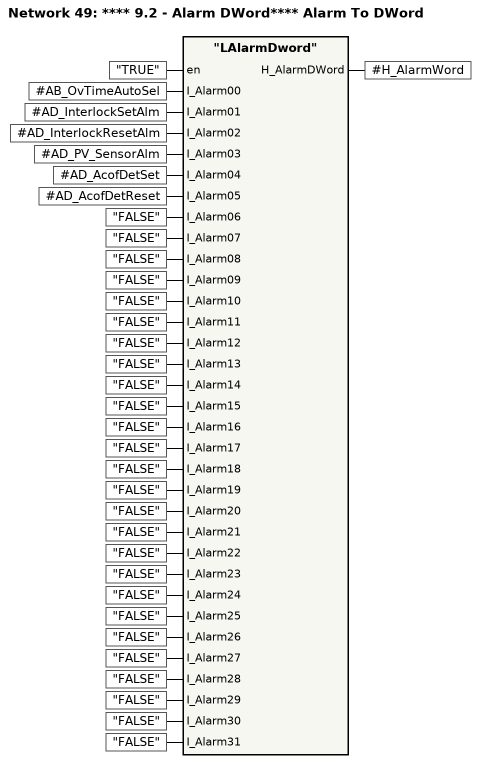
   IF "TRUE" THEN
       "LAlarmDword"(I_Alarm00 := #AB_OvTimeAutoSel,
                     I_Alarm01 := #AD_InterlockSetAlm,
                     I_Alarm02 := #AD_InterlockResetAlm,
                     I_Alarm03 := #AD_PV_SensorAlm,
                     I_Alarm04 := #AD_AcofDetSet,
                     I_Alarm05 := #AD_AcofDetReset,
                     I_Alarm06 := "FALSE",
                     I_Alarm07 := "FALSE",
                     I_Alarm08 := "FALSE",
                     I_Alarm09 := "FALSE",
                     I_Alarm10 := "FALSE",
                     I_Alarm11 := "FALSE",
                     I_Alarm12 := "FALSE",
                     I_Alarm13 := "FALSE",
                     I_Alarm14 := "FALSE",
                     I_Alarm15 := "FALSE",
                     I_Alarm16 := "FALSE",
                     I_Alarm17 := "FALSE",
                     I_Alarm18 := "FALSE",
                     I_Alarm19 := "FALSE",
                     I_Alarm20 := "FALSE",
                     I_Alarm21 := "FALSE",
                     I_Alarm22 := "FALSE",
                     I_Alarm23 := "FALSE",
                     I_Alarm24 := "FALSE",
                     I_Alarm25 := "FALSE",
                     I_Alarm26 := "FALSE",
                     I_Alarm27 := "FALSE",
                     I_Alarm28 := "FALSE",
                     I_Alarm29 := "FALSE",
                     I_Alarm30 := "FALSE",
                     I_Alarm31 := "FALSE",
                     H_AlarmDWord => #H_AlarmWord);
   END_IF;
END_REGION
END_FUNCTION_BLOCK

FUNCTION_BLOCK "LProcTimStrtStop"   // FB1735, FBD
TITLE = LProcTimeStartStop
{ S7_Optimized_Access := 'FALSE' }
AUTHOR : VCC
FAMILY : ProcEq
NAME : TimeStSt
VERSION : 1.0
// ================================================================================
// Module used to give a signal between 2 times with the calendar variable of PLC: 
// start - stop is defined by HMI
// ================================================================================
// stored: AutoNumber false, IsIECCheckEnabled false, SetENOAutomatically False, UDAEnableTagReadback false
   VAR_OUTPUT
      O_TimeActive { ExternalAccessible := 'False'; ExternalVisible := 'False'; ExternalWritable := 'False'} : Bool;   // Time active
      O_InverseTimeActive { ExternalAccessible := 'False'; ExternalVisible := 'False'; ExternalWritable := 'False'} : Bool;   // Inverse Time active
      H_IAnim { ExternalAccessible := 'False'; ExternalVisible := 'False'; ExternalWritable := 'False'} : Word;   // HMI Animation of the icon
   END_VAR
   VAR DB_SPECIFIC
      H_In : Struct   // HMI
         Start : Real := 9.0;   // Start time
         Stop : Real := 9.15;   // Stop time
      END_STRUCT;
      H_Out : Struct   // HMI
         Anim : Word;   // HMI Animation of the object
         DBnr : Int;   // HMI Animation DB number
      END_STRUCT;
      TimeActive { ExternalAccessible := 'False'; ExternalVisible := 'False'; ExternalWritable := 'False'} : Bool;   // Time active
      Start_Int { ExternalAccessible := 'False'; ExternalVisible := 'False'; ExternalWritable := 'False'} : Int := 900;   // Start integer
      Stop_Int { ExternalAccessible := 'False'; ExternalVisible := 'False'; ExternalWritable := 'False'} : Int := 915;   // Stort integer
      DBnr { ExternalAccessible := 'False'; ExternalVisible := 'False'; ExternalWritable := 'False'} : Int;   // HMI DB number
   END_VAR
BEGIN

NETWORK
TITLE = **** 1 - Inputs **** DB number
// DB number
      L     DINO;
      T     #DBnr;

NETWORK
TITLE = **** 4.4 - Machine status - Calculated **** Copy time from HMI to integer
// Copy time from HMI to integer
      L     #H_In.Start;  // Load Start time
      L     100.0;  // * 100
      *R;  // *
      RND;  // Conversion real to integer
      T     #Start_Int;  // Load start time of morning shift = Day 1

      L     #H_In.Stop;  // Load Start time of evening shift - Day 1
      L     100.0;  // * 100
      *R;  // *
      RND;  // Conversion real to integer
      T     #Stop_Int;  // Load start time of evening shift = Day 1


REGION Network 3: **** 4.4 - Machine status - Calculated **** Morning Shift of Day 1
   // Morning Shift of Day 1
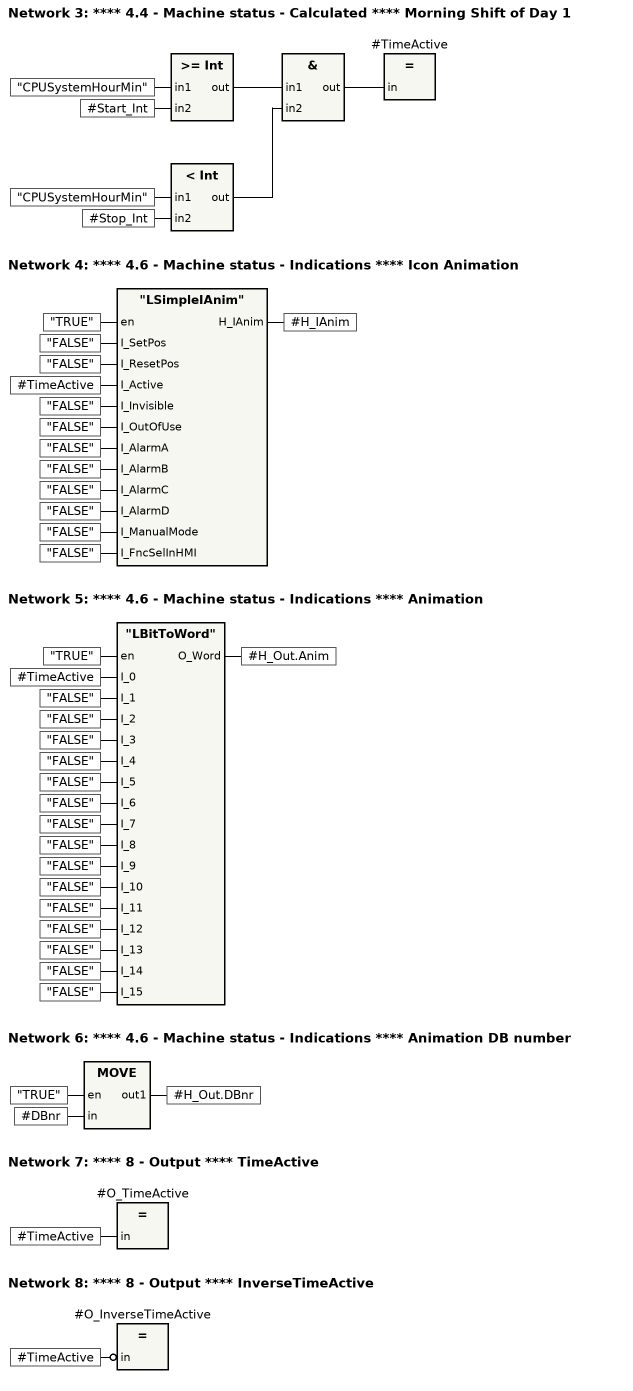
   #TimeActive := ("CPUSystemHourMin" >= #Start_Int) AND ("CPUSystemHourMin" < #Stop_Int);
END_REGION

REGION Network 4: **** 4.6 - Machine status - Indications **** Icon Animation
   // Icon Animation for HMI
   IF "TRUE" THEN
       "LSimpleIAnim"(I_SetPos := "FALSE",
                      I_ResetPos := "FALSE",
                      I_Active := #TimeActive,
                      I_Invisible := "FALSE",
                      I_OutOfUse := "FALSE",
                      I_AlarmA := "FALSE",
                      I_AlarmB := "FALSE",
                      I_AlarmC := "FALSE",
                      I_AlarmD := "FALSE",
                      I_ManualMode := "FALSE",
                      I_FncSelInHMI := "FALSE",
                      H_IAnim => #H_IAnim);
   END_IF;
END_REGION

REGION Network 5: **** 4.6 - Machine status - Indications **** Animation
   // Animation for HMI
   IF "TRUE" THEN
       "LBitToWord"(I_0 := #TimeActive,
                    I_1 := "FALSE",
                    I_2 := "FALSE",
                    I_3 := "FALSE",
                    I_4 := "FALSE",
                    I_5 := "FALSE",
                    I_6 := "FALSE",
                    I_7 := "FALSE",
                    I_8 := "FALSE",
                    I_9 := "FALSE",
                    I_10 := "FALSE",
                    I_11 := "FALSE",
                    I_12 := "FALSE",
                    I_13 := "FALSE",
                    I_14 := "FALSE",
                    I_15 := "FALSE",
                    O_Word => #H_Out.Anim);
   END_IF;
END_REGION

REGION Network 6: **** 4.6 - Machine status - Indications **** Animation DB number
   // Animation DB number
   IF "TRUE" THEN #H_Out.DBnr := #DBnr; END_IF;
END_REGION

REGION Network 7: **** 8 - Output **** TimeActive
   // TimeActive
   #O_TimeActive := #TimeActive;
END_REGION

REGION Network 8: **** 8 - Output **** InverseTimeActive
   // InverseTimeActive
   #O_InverseTimeActive := NOT #TimeActive;
END_REGION
END_FUNCTION_BLOCK

FUNCTION_BLOCK "LProcGeneralFunc"   // FB1738, FBD
TITLE = LProcGeneralFunc
{ S7_Optimized_Access := 'TRUE' }
AUTHOR : VCC
FAMILY : Control
NAME : Genfunc
VERSION : 0.1
// ================================================================================
// This module handles General Reverse Switch, General High Speed and Lamptest.
// It will also give the user and 8 bit interface for project specific functions.
// ================================================================================
// stored: AutoNumber false, IsIECCheckEnabled false, IsRetainMemResEnabled false, MemoryReserve 100, SetENOAutomatically False, UDAEnableTagReadback false
   VAR_INPUT
      I_GenRevSw { ExternalAccessible := 'False'; ExternalVisible := 'False'; ExternalWritable := 'False'} : Bool;   // General reverse switch
      I_GenHighSpeed { ExternalAccessible := 'False'; ExternalVisible := 'False'; ExternalWritable := 'False'} : Bool;   // General high speed
      I_Lamptest { ExternalAccessible := 'False'; ExternalVisible := 'False'; ExternalWritable := 'False'} : Bool;   // Lamptest PB
      I_ManualMode { ExternalAccessible := 'False'; ExternalVisible := 'False'; ExternalWritable := 'False'} : Bool := TRUE;   // Manual mode active
      I_LamptestSec { ExternalAccessible := 'False'; ExternalVisible := 'False'; ExternalWritable := 'False'} : Int := 60;   // The number of seconds that Lamptest will be on (Sec)
   END_VAR
   VAR_OUTPUT
      O_GeneralFunc : Word;   // General functions
      O_Lamptest { ExternalAccessible := 'False'; ExternalVisible := 'False'; ExternalWritable := 'False'} : Bool;   // Lamptest
      O_LamptestSteady { ExternalAccessible := 'False'; ExternalVisible := 'False'; ExternalWritable := 'False'} : Bool;   // Lamptest always on
      O_GenHighSpeed { ExternalAccessible := 'False'; ExternalVisible := 'False'; ExternalWritable := 'False'} : Bool;   // General High Speed
      O_GenRevSwitch { ExternalAccessible := 'False'; ExternalVisible := 'False'; ExternalWritable := 'False'} : Bool;   // Reverse Switch
      O_GenReverseAlarm { ExternalAccessible := 'False'; ExternalVisible := 'False'; ExternalWritable := 'False'} : Bool;   // Alarm when general reverse switch is ON while NOT in Manual mode
   END_VAR
   VAR DB_SPECIFIC
      H_HMIGenFuncCmd : Word;   // General function commands from HMI
      AutoMode { ExternalAccessible := 'False'; ExternalVisible := 'False'; ExternalWritable := 'False'} : Bool;   // Auto mode
      AutoSel { ExternalAccessible := 'False'; ExternalVisible := 'False'; ExternalWritable := 'False'} : Bool;   // Auto is selected
      AlarmAB { ExternalAccessible := 'False'; ExternalVisible := 'False'; ExternalWritable := 'False'} : Bool;   // Alarm A or B is active
      HMIGenHighSpeed { ExternalAccessible := 'False'; ExternalVisible := 'False'; ExternalWritable := 'False'} : Bool;   // General High Speed for manual movement
      HMILamptest { ExternalAccessible := 'False'; ExternalVisible := 'False'; ExternalWritable := 'False'} : Bool;   // Lamptest
      GenHighSpeedSelected { ExternalAccessible := 'False'; ExternalVisible := 'False'; ExternalWritable := 'False'} : Bool;   // General high speed is selected
      LamptestSelected : Bool;   // Lamptest is selected
      PulseLamptest { ExternalAccessible := 'False'; ExternalVisible := 'False'; ExternalWritable := 'False'} : Bool;   // Pulse for lamptest
      PulseGenHighSpeed { ExternalAccessible := 'False'; ExternalVisible := 'False'; ExternalWritable := 'False'} : Bool;   // Pulse General high speed
      TimerLamptest { ExternalAccessible := 'False'; ExternalVisible := 'False'; ExternalWritable := 'False'} : Bool;   // Timer for Lamptest
      LamptestSec { ExternalAccessible := 'False'; ExternalVisible := 'False'; ExternalWritable := 'False'} : DInt;   // Lamptest on for xxx milliesec
      LamptestMillieSec { ExternalAccessible := 'False'; ExternalVisible := 'False'; ExternalWritable := 'False'} : DInt;   // Converted value
   END_VAR
   VAR
      TimerLampTestSel { ExternalAccessible := 'False'; ExternalVisible := 'False'; ExternalWritable := 'False'; S7_SetPoint := 'True'} : "LTimer";
   END_VAR
   VAR_TEMP
      SetLamptest : Bool;   // Set Lamptest
      ResetLamptest : Bool;   // Reset Lamptest
      ElapseTime : DInt;   // Elapse time for Lamptest
   END_VAR
   VAR_TEMP   // added for the SCL form of the ladder/FBD networks
      _w1 : Bool;
      _w2 : Bool;
   END_VAR
BEGIN

REGION Network 1: **** 1 - Inputs **** Extract the general functions from HMI
   // Extract the general functions from HMI
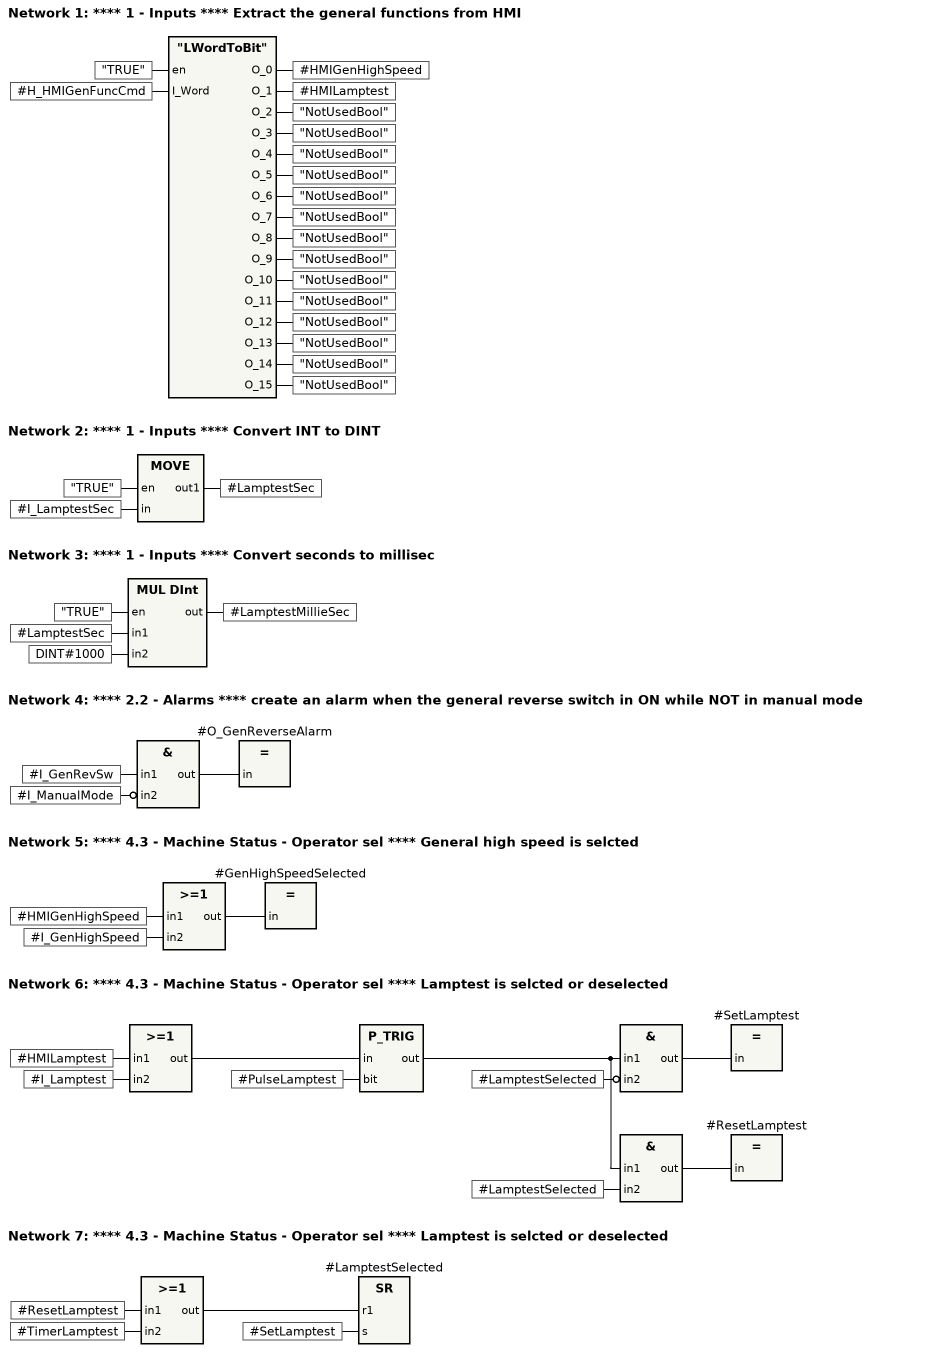
   IF "TRUE" THEN
       "LWordToBit"(I_Word := #H_HMIGenFuncCmd,
                    O_0 => #HMIGenHighSpeed,
                    O_1 => #HMILamptest,
                    O_2 => "NotUsedBool",
                    O_3 => "NotUsedBool",
                    O_4 => "NotUsedBool",
                    O_5 => "NotUsedBool",
                    O_6 => "NotUsedBool",
                    O_7 => "NotUsedBool",
                    O_8 => "NotUsedBool",
                    O_9 => "NotUsedBool",
                    O_10 => "NotUsedBool",
                    O_11 => "NotUsedBool",
                    O_12 => "NotUsedBool",
                    O_13 => "NotUsedBool",
                    O_14 => "NotUsedBool",
                    O_15 => "NotUsedBool");
   END_IF;
END_REGION

REGION Network 2: **** 1 - Inputs **** Convert INT to DINT
   // Convert INT to DINT
   IF "TRUE" THEN #LamptestSec := #I_LamptestSec; END_IF;
END_REGION

REGION Network 3: **** 1 - Inputs **** Convert seconds to millisec
   // Convert seconds to millisec
   IF "TRUE" THEN #LamptestMillieSec := #LamptestSec * DINT#1000; END_IF;
END_REGION

REGION Network 4: **** 2.2 - Alarms **** create an alarm when the general reverse switch in ON while NOT in manual mode
   // create an alarm when the general reverse switch in ON while NOT in manual mode
   #O_GenReverseAlarm := #I_GenRevSw AND NOT #I_ManualMode;
END_REGION

REGION Network 5: **** 4.3 - Machine Status - Operator sel **** General high speed is selcted
   // General high speed is selcted
   #GenHighSpeedSelected := #HMIGenHighSpeed OR #I_GenHighSpeed;
END_REGION

REGION Network 6: **** 4.3 - Machine Status - Operator sel **** Lamptest is selcted or deselected
   // Lamptest is selcted or deselected
   #_w1 := #HMILamptest OR #I_Lamptest;
   #_w2 := #_w1 AND NOT #PulseLamptest;   // rising edge
   #PulseLamptest := #_w1;
   #SetLamptest := #_w2 AND NOT #LamptestSelected;
   #ResetLamptest := #_w2 AND #LamptestSelected;
END_REGION

REGION Network 7: **** 4.3 - Machine Status - Operator sel **** Lamptest is selcted or deselected
   // Lamptest is selcted or deselected
   IF #SetLamptest THEN
       #LamptestSelected := TRUE;   // SR flip-flop
   END_IF;
   IF #ResetLamptest OR #TimerLamptest THEN #LamptestSelected := FALSE; END_IF;
END_REGION

REGION Network 8: **** 4.3 - Machine Status - Operator sel **** Timer for Lamptest
   // Timer for Lamptest
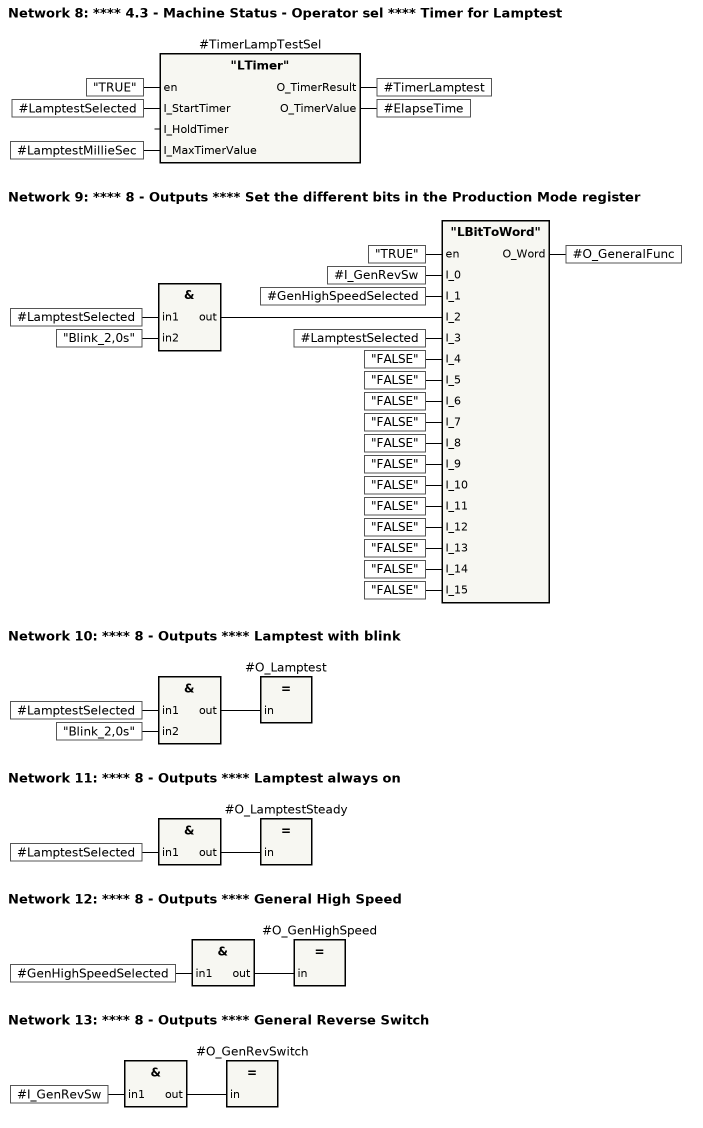
   IF "TRUE" THEN
       #TimerLampTestSel(I_StartTimer := #LamptestSelected,   // "LTimer"
                         I_MaxTimerValue := #LamptestMillieSec,
                         O_TimerResult => #TimerLamptest,
                         O_TimerValue => #ElapseTime);
   END_IF;
END_REGION

REGION Network 9: **** 8 - Outputs **** Set the different bits in the Production Mode register
   // Set the different bits in the Production Mode register
   IF "TRUE" THEN
       "LBitToWord"(I_0 := #I_GenRevSw,
                    I_1 := #GenHighSpeedSelected,
                    I_2 := #LamptestSelected AND "Blink_2,0s",
                    I_3 := #LamptestSelected,
                    I_4 := "FALSE",
                    I_5 := "FALSE",
                    I_6 := "FALSE",
                    I_7 := "FALSE",
                    I_8 := "FALSE",
                    I_9 := "FALSE",
                    I_10 := "FALSE",
                    I_11 := "FALSE",
                    I_12 := "FALSE",
                    I_13 := "FALSE",
                    I_14 := "FALSE",
                    I_15 := "FALSE",
                    O_Word => #O_GeneralFunc);
   END_IF;
END_REGION

REGION Network 10: **** 8 - Outputs **** Lamptest with blink
   // Lamptest with blink
   #O_Lamptest := #LamptestSelected AND "Blink_2,0s";
END_REGION

REGION Network 11: **** 8 - Outputs **** Lamptest always on
   // Lamptest always on
   #O_LamptestSteady := #LamptestSelected;
END_REGION

REGION Network 12: **** 8 - Outputs **** General High Speed
   // General High Speed
   #O_GenHighSpeed := #GenHighSpeedSelected;
END_REGION

REGION Network 13: **** 8 - Outputs **** General Reverse Switch
   // General Reverse Switch
   #O_GenRevSwitch := #I_GenRevSw;
END_REGION
END_FUNCTION_BLOCK

FUNCTION_BLOCK "LProcPAC"   // FB1740, FBD
TITLE = LProcPAC
{ S7_Optimized_Access := 'TRUE' }
AUTHOR : CSTAAL
VERSION : 0.1
// This module handles the power measuring device
// stored: AutoNumber false, IsIECCheckEnabled false, IsRetainMemResEnabled false, MemoryReserve 100, SetENOAutomatically False, UDAEnableTagReadback false
   VAR_INPUT
      I_HWSubModule { ExternalAccessible := 'False'; ExternalVisible := 'False'; ExternalWritable := 'False'} : HW_SUBMODULE;   // Connection with Hardware Sub Module
   END_VAR
   VAR_OUTPUT
      O_ControlBytes { ExternalAccessible := 'False'; ExternalVisible := 'False'; ExternalWritable := 'False'} : Word;   // Control Bytes for the PAC
      O_AlarmA { ExternalAccessible := 'False'; ExternalVisible := 'False'; ExternalWritable := 'False'} : Bool;   // Alarm A
      O_AlarmB { ExternalAccessible := 'False'; ExternalVisible := 'False'; ExternalWritable := 'False'} : Bool;   // Alarm B
      O_AlarmC { ExternalAccessible := 'False'; ExternalVisible := 'False'; ExternalWritable := 'False'} : Bool;   // Alarm C
      O_AlarmD { ExternalAccessible := 'False'; ExternalVisible := 'False'; ExternalWritable := 'False'} : Bool;   // Alarm D
      O_AlarmABCondition { ExternalAccessible := 'False'; ExternalVisible := 'False'; ExternalWritable := 'False'} : Bool;   // Alarms resetable
      H_IAnim { ExternalAccessible := 'False'; ExternalVisible := 'False'; ExternalWritable := 'False'} : Word;   // Animation bits to Icon in WinCC
      H_AlarmWord { ExternalAccessible := 'False'; ExternalVisible := 'False'; ExternalWritable := 'False'} : DWord;   // Alarm Word
   END_VAR
   VAR DB_SPECIFIC
      Cmd { ExternalAccessible := 'False'; ExternalVisible := 'False'; ExternalWritable := 'False'} : Struct   // Command (copied from HMI Command) / Command
         Reset_min_max_Data { ExternalAccessible := 'False'; ExternalVisible := 'False'; ExternalWritable := 'False'} : Bool := FALSE;   // 0 / Reset_min_max_Data
         Reset_Energy_Meter { ExternalAccessible := 'False'; ExternalVisible := 'False'; ExternalWritable := 'False'} : Bool := FALSE;   // 1 / Reset_Energy_Meter
      END_STRUCT;
   END_VAR
   VAR
      C_UnitAmps { ExternalAccessible := 'False'; ExternalVisible := 'False'; ExternalWritable := 'False'} : Int;   // Unit Amps (1 = mA; 2 = kA)
      C_UnitVolts { ExternalAccessible := 'False'; ExternalVisible := 'False'; ExternalWritable := 'False'} : Int;   // Unit Volts (1 = mV; 2 = V)
      C_UnitWatts { ExternalAccessible := 'False'; ExternalVisible := 'False'; ExternalWritable := 'False'} : Int;   // Unit Watts (1 = W; 2 = kW)
      Units { ExternalAccessible := 'False'; ExternalVisible := 'False'; ExternalWritable := 'False'} : Struct   // Units
         "Amps-mA" { ExternalAccessible := 'False'; ExternalVisible := 'False'; ExternalWritable := 'False'} : Bool;   // Amps in mA
         "Amps-kA" { ExternalAccessible := 'False'; ExternalVisible := 'False'; ExternalWritable := 'False'} : Bool;   // Amps in kA
         "Volts-mV" { ExternalAccessible := 'False'; ExternalVisible := 'False'; ExternalWritable := 'False'} : Bool;   // Volts in mV
         "Volts-kV" { ExternalAccessible := 'False'; ExternalVisible := 'False'; ExternalWritable := 'False'} : Bool;   // Volts in kV
         "Watts-W" { ExternalAccessible := 'False'; ExternalVisible := 'False'; ExternalWritable := 'False'} : Bool;   // Watts in W
         "Watts-kW" { ExternalAccessible := 'False'; ExternalVisible := 'False'; ExternalWritable := 'False'} : Bool;   // Watts in kW
      END_STRUCT;
      H_HMICmd : Word;   // HMI Command
   END_VAR
   VAR DB_SPECIFIC
      H_Out : Struct   // HMI
         Anim : Word;   // HMI Animation of the object
         DBnr : Int;   // HMI Animation DB number
         U12 : Real;   // Voltage L1-L2
         U23 : Real;   // Voltage L2-L3
         U31 : Real;   // Voltage L3-L1
         U12Max : Real;   // MAX Voltage L1-L2
         U23Max : Real;   // MAX Voltage L2-L3
         U31Max : Real;   // MAX Voltage L3-L1
         UL1 : Real;   // UL1
         UL2 : Real;   // UL2
         UL3 : Real;   // UL3
         UL1Max : Real;   // MAX Voltage L1
         UL2Max : Real;   // MAX Voltage L2
         UL3Max : Real;   // MAX Voltage L3
         I1 : Real;   // Current L1
         I2 : Real;   // Current L2
         I3 : Real;   // Current L3
         I1Max : Real;   // MAX Current L1
         I2Max : Real;   // MAX Current L2
         I3Max : Real;   // MAX Current L3
         PTotal : Real;   // Total active power
         PTotalMax : Real;   // Total MAX active power
      END_STRUCT;
   END_VAR
   VAR
      AlarmA { ExternalAccessible := 'False'; ExternalVisible := 'False'; ExternalWritable := 'False'} : Bool;   // Alarm A
      AlarmB { ExternalAccessible := 'False'; ExternalVisible := 'False'; ExternalWritable := 'False'} : Bool;   // Alarm B
      AlarmC { ExternalAccessible := 'False'; ExternalVisible := 'False'; ExternalWritable := 'False'} : Bool;   // Alarm C
      AlarmD { ExternalAccessible := 'False'; ExternalVisible := 'False'; ExternalWritable := 'False'} : Bool;   // Alarm D
      AlarmABCondition { ExternalAccessible := 'False'; ExternalVisible := 'False'; ExternalWritable := 'False'} : Bool;   // Alarm AB condition
   END_VAR
   VAR DB_SPECIFIC
      DBnr { ExternalAccessible := 'False'; ExternalVisible := 'False'; ExternalWritable := 'False'} : Int;   // HMI DB number
   END_VAR
   VAR
      _PACDriver { ExternalAccessible := 'False'; ExternalVisible := 'False'; ExternalWritable := 'False'} : "LProcPAC-Driver";   // FB
      _PACVisu { ExternalAccessible := 'False'; ExternalVisible := 'False'; ExternalWritable := 'False'} : "LProcPAC-Visu";   // FB
   END_VAR
   VAR_TEMP
      ControlBytes : Word;   // Control Bytes for the PAC
      L12 : Real;   // Temporary test variable
      L23 : Real;   // Temporary test variable
      L31 : Real;   // Temporary test variable
   END_VAR
   VAR_TEMP   // added for the SCL form of the ladder/FBD networks
      _w1 : Bool;
   END_VAR
BEGIN

NETWORK
TITLE = **** 1 - Inputs **** DB number
// DB number
      L     DINO;
      T     #DBnr;

REGION Network 2: **** 1 - Inputs **** HMI Commands
   // HMI Commands
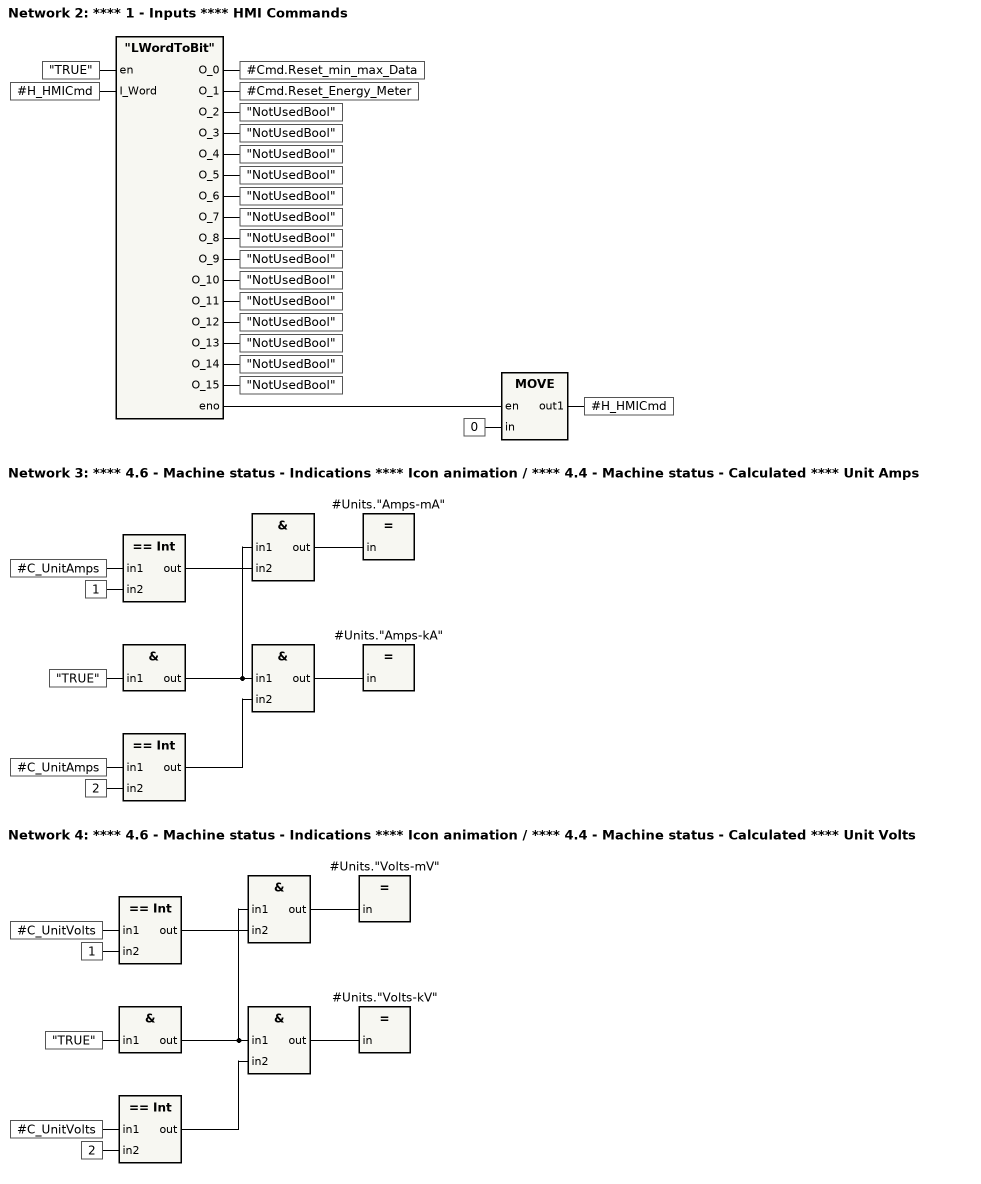
   "LWordToBit"(EN := "TRUE",
                I_Word := #H_HMICmd,
                O_0 => #Cmd.Reset_min_max_Data,
                O_1 => #Cmd.Reset_Energy_Meter,
                O_2 => "NotUsedBool",
                O_3 => "NotUsedBool",
                O_4 => "NotUsedBool",
                O_5 => "NotUsedBool",
                O_6 => "NotUsedBool",
                O_7 => "NotUsedBool",
                O_8 => "NotUsedBool",
                O_9 => "NotUsedBool",
                O_10 => "NotUsedBool",
                O_11 => "NotUsedBool",
                O_12 => "NotUsedBool",
                O_13 => "NotUsedBool",
                O_14 => "NotUsedBool",
                O_15 => "NotUsedBool",
                ENO => #_w1);
   IF #_w1 THEN #H_HMICmd := 0; END_IF;
END_REGION

REGION Network 3: **** 4.6 - Machine status - Indications **** Icon animation / **** 4.4 - Machine status - Calculated **** Unit Amps
   // Icon animation to WinCC / Unit Amps
   #Units."Amps-mA" := "TRUE" AND (#C_UnitAmps = 1);
   #Units."Amps-kA" := "TRUE" AND (#C_UnitAmps = 2);
END_REGION

REGION Network 4: **** 4.6 - Machine status - Indications **** Icon animation / **** 4.4 - Machine status - Calculated **** Unit Volts
   // Icon animation to WinCC / Unit Volts
   #Units."Volts-mV" := "TRUE" AND (#C_UnitVolts = 1);
   #Units."Volts-kV" := "TRUE" AND (#C_UnitVolts = 2);
END_REGION

REGION Network 5: **** 4.6 - Machine status - Indications **** Icon animation / **** 4.4 - Machine status - Calculated **** Unit Watts
   // Icon animation to WinCC / Unit Watts
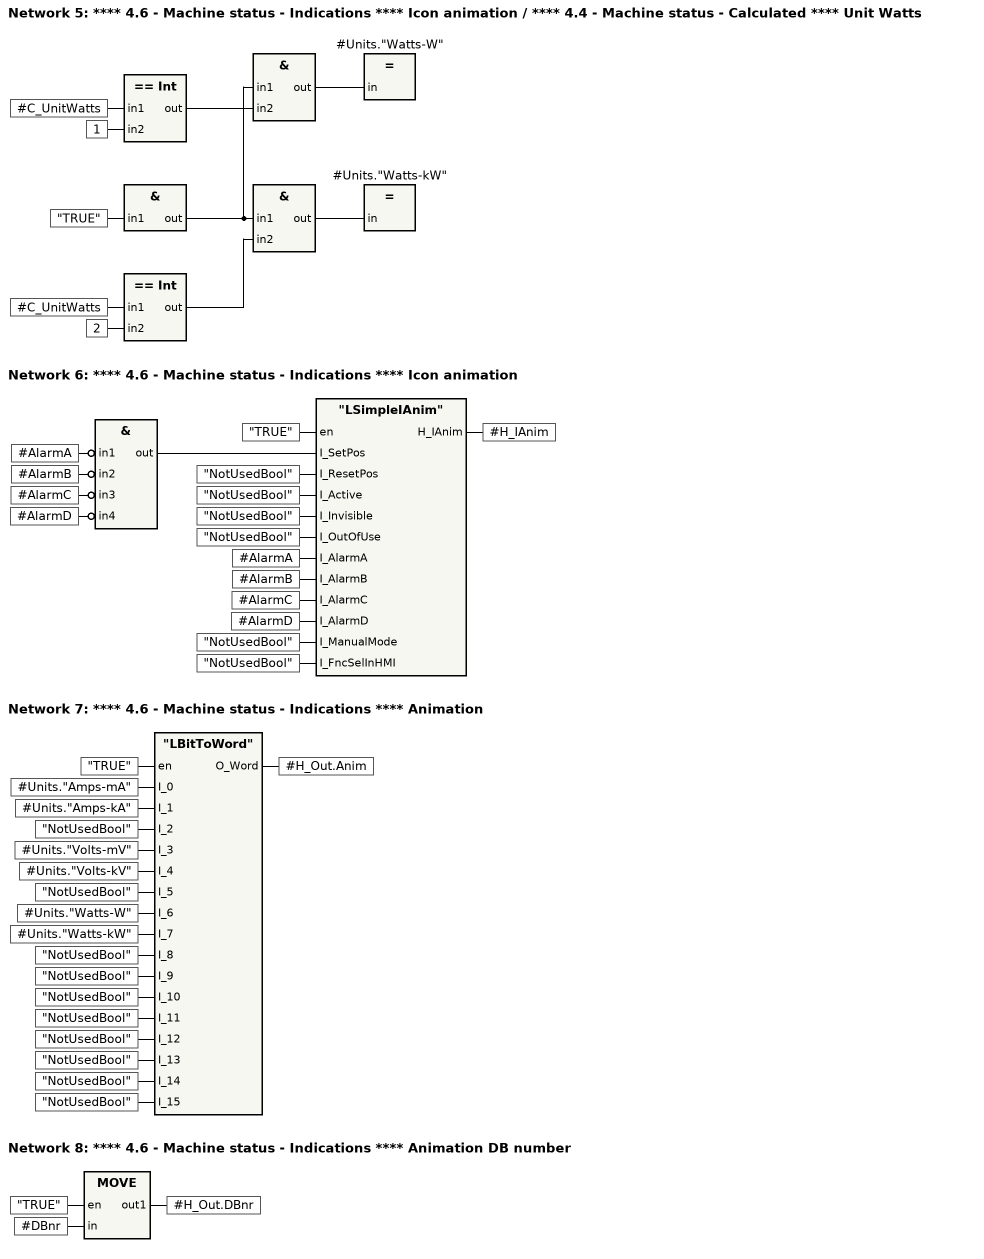
   #Units."Watts-W" := "TRUE" AND (#C_UnitWatts = 1);
   #Units."Watts-kW" := "TRUE" AND (#C_UnitWatts = 2);
END_REGION

REGION Network 6: **** 4.6 - Machine status - Indications **** Icon animation
   // Icon animation to WinCC / Icon animation
   IF "TRUE" THEN
       "LSimpleIAnim"(I_SetPos := NOT #AlarmA AND NOT #AlarmB AND NOT #AlarmC AND NOT #AlarmD,
                      I_ResetPos := "NotUsedBool",
                      I_Active := "NotUsedBool",
                      I_Invisible := "NotUsedBool",
                      I_OutOfUse := "NotUsedBool",
                      I_AlarmA := #AlarmA,
                      I_AlarmB := #AlarmB,
                      I_AlarmC := #AlarmC,
                      I_AlarmD := #AlarmD,
                      I_ManualMode := "NotUsedBool",
                      I_FncSelInHMI := "NotUsedBool",
                      H_IAnim => #H_IAnim);
   END_IF;
END_REGION

REGION Network 7: **** 4.6 - Machine status - Indications **** Animation
   // Animation
   IF "TRUE" THEN
       "LBitToWord"(I_0 := #Units."Amps-mA",
                    I_1 := #Units."Amps-kA",
                    I_2 := "NotUsedBool",
                    I_3 := #Units."Volts-mV",
                    I_4 := #Units."Volts-kV",
                    I_5 := "NotUsedBool",
                    I_6 := #Units."Watts-W",
                    I_7 := #Units."Watts-kW",
                    I_8 := "NotUsedBool",
                    I_9 := "NotUsedBool",
                    I_10 := "NotUsedBool",
                    I_11 := "NotUsedBool",
                    I_12 := "NotUsedBool",
                    I_13 := "NotUsedBool",
                    I_14 := "NotUsedBool",
                    I_15 := "NotUsedBool",
                    O_Word => #H_Out.Anim);
   END_IF;
END_REGION

REGION Network 8: **** 4.6 - Machine status - Indications **** Animation DB number
   // Animation DB number
   IF "TRUE" THEN #H_Out.DBnr := #DBnr; END_IF;
END_REGION

REGION Network 9: **** 7.1 SubModules - Non Machine **** Method 2: PAC3200 Driver
   // PAC3200 Driver
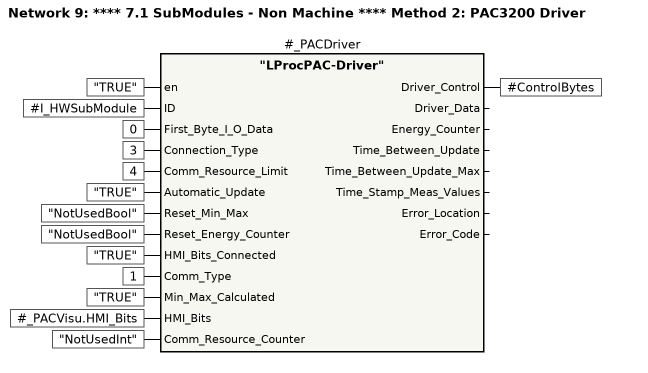
   IF "TRUE" THEN
       #_PACDriver(ID := #I_HWSubModule,   // "LProcPAC-Driver"
                   First_Byte_I_O_Data := 0,
                   Connection_Type := 3,
                   Comm_Resource_Limit := 4,
                   Automatic_Update := "TRUE",
                   Reset_Min_Max := "NotUsedBool",
                   Reset_Energy_Counter := "NotUsedBool",
                   HMI_Bits_Connected := "TRUE",
                   Comm_Type := 1,
                   Min_Max_Calculated := "TRUE",
                   HMI_Bits := #_PACVisu.HMI_Bits,
                   Comm_Resource_Counter := "NotUsedInt",
                   Driver_Control => #ControlBytes);
   END_IF;
END_REGION

REGION Network 10: **** 7.1 SubModules - Non Machine **** Method 2: PAC3200 Visualisation
   // PAC3200 Visualisation
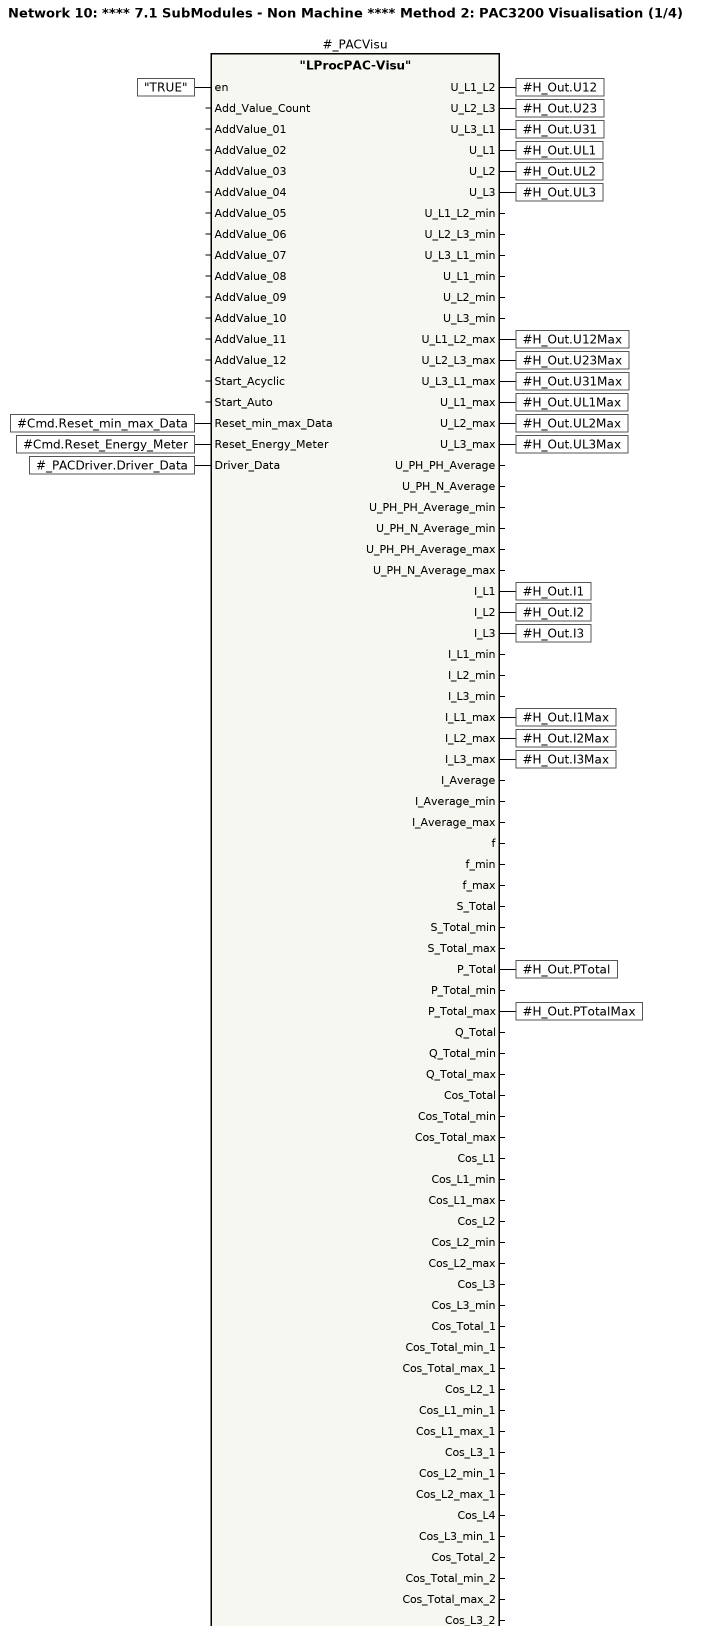
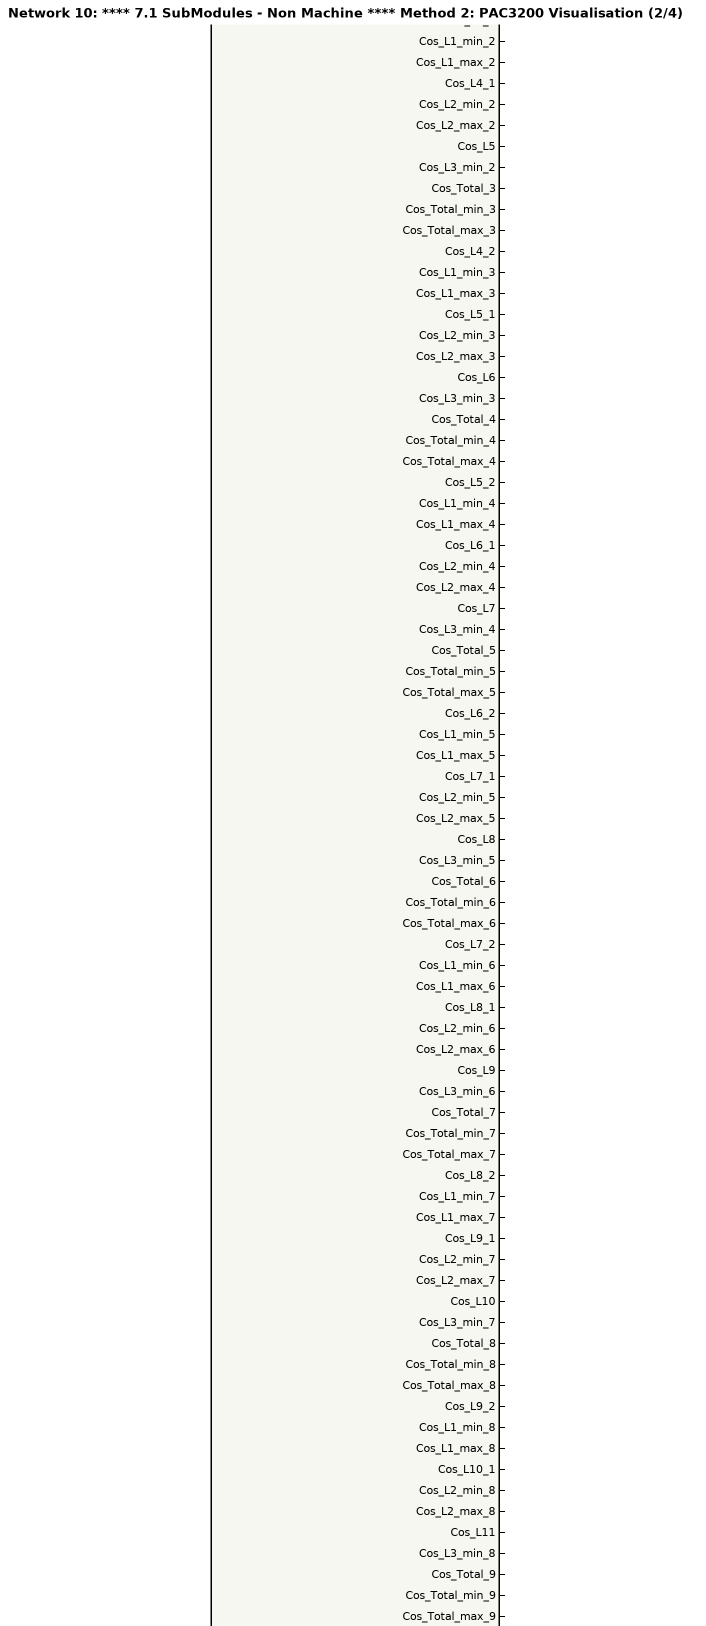
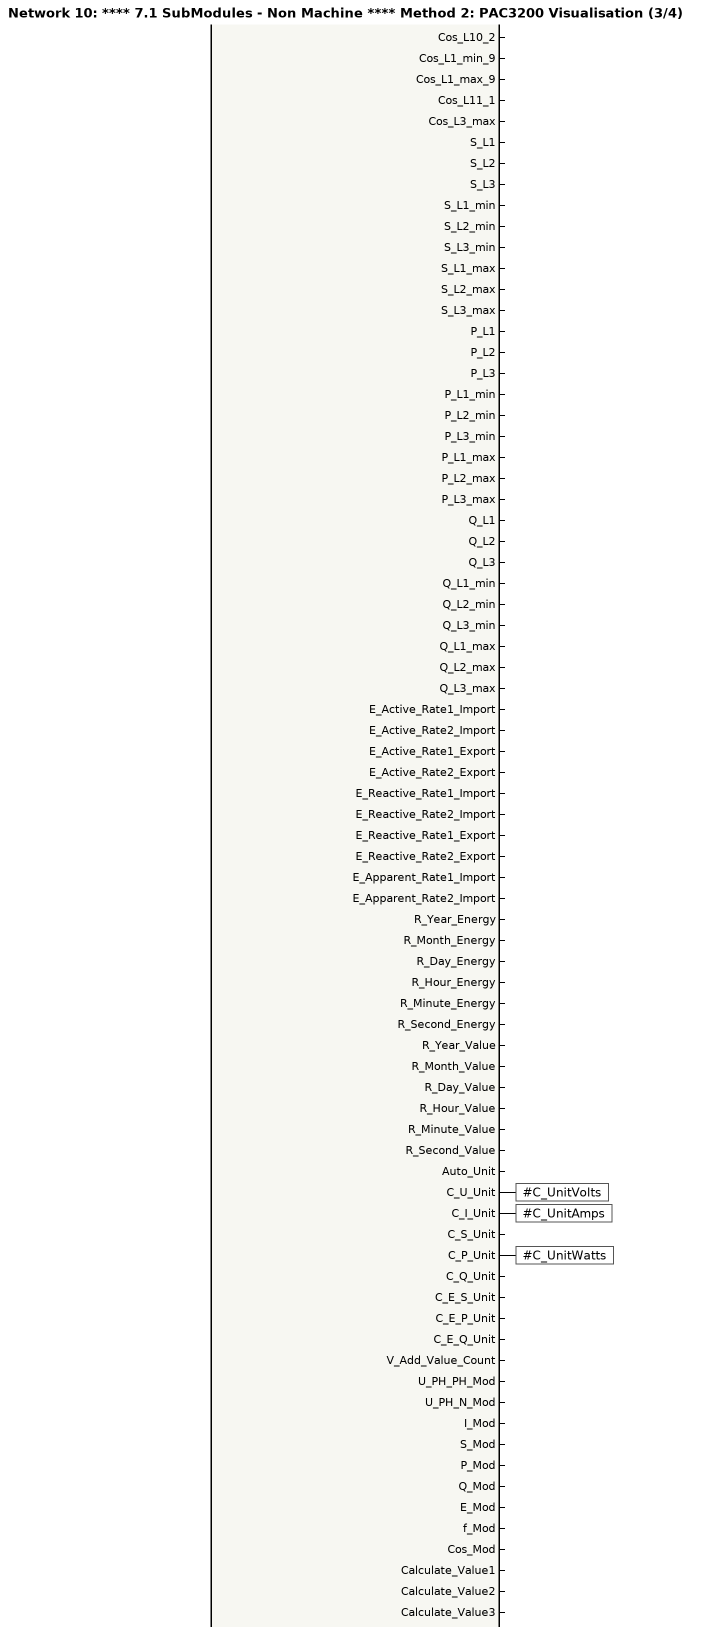
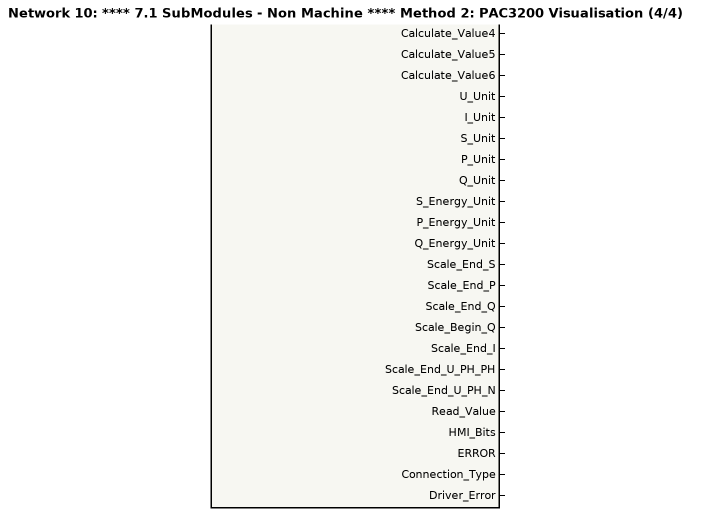
   IF "TRUE" THEN
       #_PACVisu(Reset_min_max_Data := #Cmd.Reset_min_max_Data,   // "LProcPAC-Visu"
                 Reset_Energy_Meter := #Cmd.Reset_Energy_Meter,
                 Driver_Data := #_PACDriver.Driver_Data,
                 U_L1_L2 => #H_Out.U12,
                 U_L2_L3 => #H_Out.U23,
                 U_L3_L1 => #H_Out.U31,
                 U_L1 => #H_Out.UL1,
                 U_L2 => #H_Out.UL2,
                 U_L3 => #H_Out.UL3,
                 U_L1_L2_max => #H_Out.U12Max,
                 U_L2_L3_max => #H_Out.U23Max,
                 U_L3_L1_max => #H_Out.U31Max,
                 U_L1_max => #H_Out.UL1Max,
                 U_L2_max => #H_Out.UL2Max,
                 U_L3_max => #H_Out.UL3Max,
                 I_L1 => #H_Out.I1,
                 I_L2 => #H_Out.I2,
                 I_L3 => #H_Out.I3,
                 I_L1_max => #H_Out.I1Max,
                 I_L2_max => #H_Out.I2Max,
                 I_L3_max => #H_Out.I3Max,
                 P_Total => #H_Out.PTotal,
                 P_Total_max => #H_Out.PTotalMax,
                 C_U_Unit => #C_UnitVolts,
                 C_I_Unit => #C_UnitAmps,
                 C_P_Unit => #C_UnitWatts);
   END_IF;
END_REGION

REGION Network 11: *** 8 - Outputs **** Control Bytes PAC
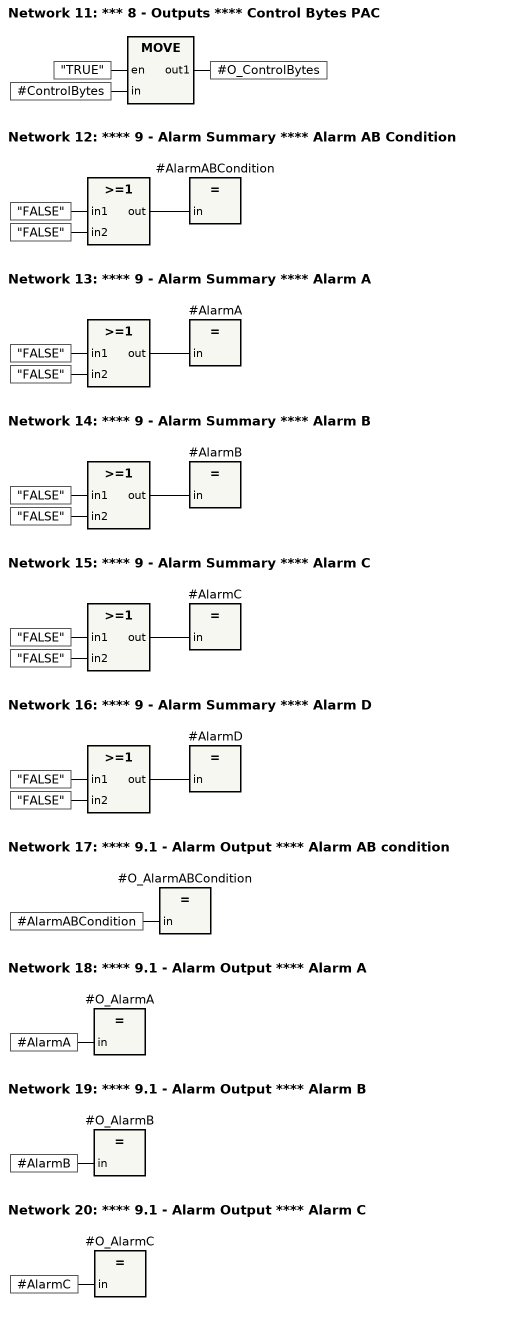
   IF "TRUE" THEN #O_ControlBytes := #ControlBytes; END_IF;
END_REGION

REGION Network 12: **** 9 - Alarm Summary **** Alarm AB Condition
   #AlarmABCondition := "FALSE" OR "FALSE";
END_REGION

REGION Network 13: **** 9 - Alarm Summary **** Alarm A
   #AlarmA := "FALSE" OR "FALSE";
END_REGION

REGION Network 14: **** 9 - Alarm Summary **** Alarm B
   #AlarmB := "FALSE" OR "FALSE";
END_REGION

REGION Network 15: **** 9 - Alarm Summary **** Alarm C
   #AlarmC := "FALSE" OR "FALSE";
END_REGION

REGION Network 16: **** 9 - Alarm Summary **** Alarm D
   #AlarmD := "FALSE" OR "FALSE";
END_REGION

REGION Network 17: **** 9.1 - Alarm Output **** Alarm AB condition
   // Alarm AB condition
   #O_AlarmABCondition := #AlarmABCondition;
END_REGION

REGION Network 18: **** 9.1 - Alarm Output **** Alarm A
   // Output Alarm A
   #O_AlarmA := #AlarmA;
END_REGION

REGION Network 19: **** 9.1 - Alarm Output **** Alarm B
   // Output Alarm B
   #O_AlarmB := #AlarmB;
END_REGION

REGION Network 20: **** 9.1 - Alarm Output **** Alarm C
   // Output Alarm A
   #O_AlarmC := #AlarmC;
END_REGION

REGION Network 21: **** 9.1 - Alarm Output **** Alarm D
   // Output Alarm D
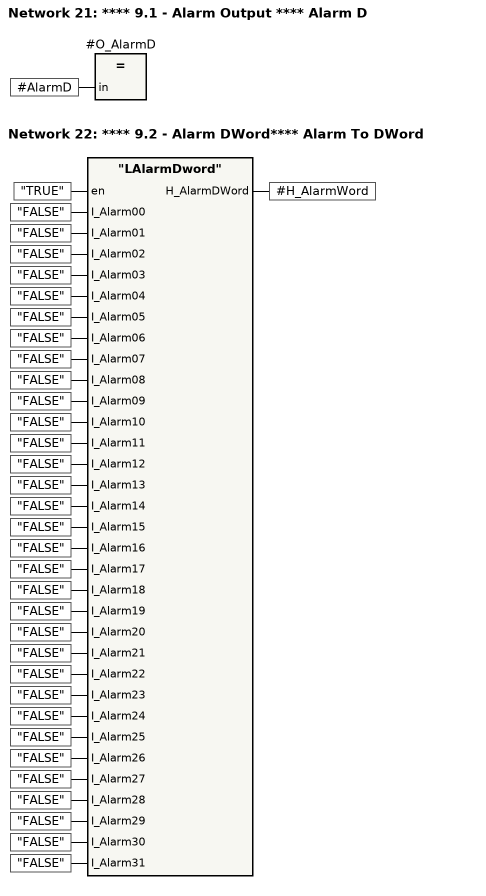
   #O_AlarmD := #AlarmD;
END_REGION

REGION Network 22: **** 9.2 - Alarm DWord**** Alarm To DWord
   // Alarm Word
   IF "TRUE" THEN
       "LAlarmDword"(I_Alarm00 := "FALSE",
                     I_Alarm01 := "FALSE",
                     I_Alarm02 := "FALSE",
                     I_Alarm03 := "FALSE",
                     I_Alarm04 := "FALSE",
                     I_Alarm05 := "FALSE",
                     I_Alarm06 := "FALSE",
                     I_Alarm07 := "FALSE",
                     I_Alarm08 := "FALSE",
                     I_Alarm09 := "FALSE",
                     I_Alarm10 := "FALSE",
                     I_Alarm11 := "FALSE",
                     I_Alarm12 := "FALSE",
                     I_Alarm13 := "FALSE",
                     I_Alarm14 := "FALSE",
                     I_Alarm15 := "FALSE",
                     I_Alarm16 := "FALSE",
                     I_Alarm17 := "FALSE",
                     I_Alarm18 := "FALSE",
                     I_Alarm19 := "FALSE",
                     I_Alarm20 := "FALSE",
                     I_Alarm21 := "FALSE",
                     I_Alarm22 := "FALSE",
                     I_Alarm23 := "FALSE",
                     I_Alarm24 := "FALSE",
                     I_Alarm25 := "FALSE",
                     I_Alarm26 := "FALSE",
                     I_Alarm27 := "FALSE",
                     I_Alarm28 := "FALSE",
                     I_Alarm29 := "FALSE",
                     I_Alarm30 := "FALSE",
                     I_Alarm31 := "FALSE",
                     H_AlarmDWord => #H_AlarmWord);
   END_IF;
END_REGION
END_FUNCTION_BLOCK

FUNCTION_BLOCK "LProcPAC-Driver"   // FB1741, SCL
TITLE = LProcPAC-Driver
{ S7_Optimized_Access := 'FALSE' }
AUTHOR : CSTAAL
VERSION : 2.0
// stored: AutoNumber false, IsIECCheckEnabled false, SetENOAutomatically False, UDAEnableTagReadback false
   VAR_INPUT
      ID { ExternalAccessible := 'False'; ExternalVisible := 'False'; ExternalWritable := 'False'} : HW_IO := 0;   // PROFINET = The diagnostic address of the SENTRON PAC; PROFIBUS = The number of the first byte of the input data of the PAC.
      First_Byte_I_O_Data { ExternalAccessible := 'False'; ExternalVisible := 'False'; ExternalWritable := 'False'} : Int := 0;   // The number of the first byte of the control bytes of the SENTRON PAC.
      Connection_Type { ExternalAccessible := 'False'; ExternalVisible := 'False'; ExternalWritable := 'False'} : Int := 1;   // The connection type of the Energy Meter: 1 = single phase, 3 = 3 phase
      Comm_Resource_Limit { ExternalAccessible := 'False'; ExternalVisible := 'False'; ExternalWritable := 'False'} : Int := 4;   // The limit of resources, which can be used by the drviers.
      Automatic_Update { ExternalAccessible := 'False'; ExternalVisible := 'False'; ExternalWritable := 'False'} : Bool := FALSE;   // TRUE = Always update the measurement values as fast as possible.
      Reset_Min_Max { ExternalAccessible := 'False'; ExternalVisible := 'False'; ExternalWritable := 'False'} : Bool := FALSE;   // FALSE ==> TRUE = Reset the minimum and maximum values.
      Reset_Energy_Counter { ExternalAccessible := 'False'; ExternalVisible := 'False'; ExternalWritable := 'False'} : Bool := FALSE;   // FALSE ==> TRUE = Reset the energy counter of the Energy Meter.
      HMI_Bits_Connected { ExternalAccessible := 'False'; ExternalVisible := 'False'; ExternalWritable := 'False'} : Bool := FALSE;   // TRUE = Structure HMI_Bits is connected; FALSE = Structure HMI_Bits is not connected
      Comm_Type { ExternalAccessible := 'False'; ExternalVisible := 'False'; ExternalWritable := 'False'} : Int := 1;   // The communication type, to the SENTRON PAC: 1 = PROFINET, 2 = PROFIBUS
      Min_Max_Calculated { ExternalAccessible := 'False'; ExternalVisible := 'False'; ExternalWritable := 'False'} : Bool := TRUE;   // Only used for PROFIBUS: TRUE = Min-Max-Values are calculated in the driver; FALSE = Min-Max-Values read from the driver.
   END_VAR
   VAR_OUTPUT
      Driver_Control { ExternalAccessible := 'False'; ExternalVisible := 'False'; ExternalWritable := 'False'} : Word;   // Driver Control
      Driver_Data { ExternalAccessible := 'False'; ExternalVisible := 'False'; ExternalWritable := 'False'} : Struct   // The structure including all measurement values. Used for the visualization and the connection to the E2M_Visu block.
         U_L1_L2 { ExternalAccessible := 'False'; ExternalVisible := 'False'; ExternalWritable := 'False'} : Real;
         U_L2_L3 { ExternalAccessible := 'False'; ExternalVisible := 'False'; ExternalWritable := 'False'} : Real;
         U_L3_L1 { ExternalAccessible := 'False'; ExternalVisible := 'False'; ExternalWritable := 'False'} : Real;
         U_L1 { ExternalAccessible := 'False'; ExternalVisible := 'False'; ExternalWritable := 'False'} : Real;
         U_L2 { ExternalAccessible := 'False'; ExternalVisible := 'False'; ExternalWritable := 'False'} : Real;
         U_L3 { ExternalAccessible := 'False'; ExternalVisible := 'False'; ExternalWritable := 'False'} : Real;
         U_L1_L2_min { ExternalAccessible := 'False'; ExternalVisible := 'False'; ExternalWritable := 'False'} : Real;
         U_L2_L3_min { ExternalAccessible := 'False'; ExternalVisible := 'False'; ExternalWritable := 'False'} : Real;
         U_L3_L1_min { ExternalAccessible := 'False'; ExternalVisible := 'False'; ExternalWritable := 'False'} : Real;
         U_L1_min { ExternalAccessible := 'False'; ExternalVisible := 'False'; ExternalWritable := 'False'} : Real;
         U_L2_min { ExternalAccessible := 'False'; ExternalVisible := 'False'; ExternalWritable := 'False'} : Real;
         U_L3_min { ExternalAccessible := 'False'; ExternalVisible := 'False'; ExternalWritable := 'False'} : Real;
         U_L1_L2_max { ExternalAccessible := 'False'; ExternalVisible := 'False'; ExternalWritable := 'False'} : Real;
         U_L2_L3_max { ExternalAccessible := 'False'; ExternalVisible := 'False'; ExternalWritable := 'False'} : Real;
         U_L3_L1_max { ExternalAccessible := 'False'; ExternalVisible := 'False'; ExternalWritable := 'False'} : Real;
         U_L1_max { ExternalAccessible := 'False'; ExternalVisible := 'False'; ExternalWritable := 'False'} : Real;
         U_L2_max { ExternalAccessible := 'False'; ExternalVisible := 'False'; ExternalWritable := 'False'} : Real;
         U_L3_max { ExternalAccessible := 'False'; ExternalVisible := 'False'; ExternalWritable := 'False'} : Real;
         U_PH_PH_Average { ExternalAccessible := 'False'; ExternalVisible := 'False'; ExternalWritable := 'False'} : Real;
         U_PH_N_Average { ExternalAccessible := 'False'; ExternalVisible := 'False'; ExternalWritable := 'False'} : Real;
         U_PH_PH_Average_min { ExternalAccessible := 'False'; ExternalVisible := 'False'; ExternalWritable := 'False'} : Real;
         U_PH_N_Average_min { ExternalAccessible := 'False'; ExternalVisible := 'False'; ExternalWritable := 'False'} : Real;
         U_PH_PH_Average_max { ExternalAccessible := 'False'; ExternalVisible := 'False'; ExternalWritable := 'False'} : Real;
         U_PH_N_Average_max { ExternalAccessible := 'False'; ExternalVisible := 'False'; ExternalWritable := 'False'} : Real;
         I_L1 { ExternalAccessible := 'False'; ExternalVisible := 'False'; ExternalWritable := 'False'} : Real;
         I_L2 { ExternalAccessible := 'False'; ExternalVisible := 'False'; ExternalWritable := 'False'} : Real;
         I_L3 { ExternalAccessible := 'False'; ExternalVisible := 'False'; ExternalWritable := 'False'} : Real;
         I_L1_min { ExternalAccessible := 'False'; ExternalVisible := 'False'; ExternalWritable := 'False'} : Real;
         I_L2_min { ExternalAccessible := 'False'; ExternalVisible := 'False'; ExternalWritable := 'False'} : Real;
         I_L3_min { ExternalAccessible := 'False'; ExternalVisible := 'False'; ExternalWritable := 'False'} : Real;
         I_L1_max { ExternalAccessible := 'False'; ExternalVisible := 'False'; ExternalWritable := 'False'} : Real;
         I_L2_max { ExternalAccessible := 'False'; ExternalVisible := 'False'; ExternalWritable := 'False'} : Real;
         I_L3_max { ExternalAccessible := 'False'; ExternalVisible := 'False'; ExternalWritable := 'False'} : Real;
         I_Average { ExternalAccessible := 'False'; ExternalVisible := 'False'; ExternalWritable := 'False'} : Real;
         I_Average_min { ExternalAccessible := 'False'; ExternalVisible := 'False'; ExternalWritable := 'False'} : Real;
         I_Average_max { ExternalAccessible := 'False'; ExternalVisible := 'False'; ExternalWritable := 'False'} : Real;
         f { ExternalAccessible := 'False'; ExternalVisible := 'False'; ExternalWritable := 'False'} : Real;
         f_min { ExternalAccessible := 'False'; ExternalVisible := 'False'; ExternalWritable := 'False'} : Real;
         f_max { ExternalAccessible := 'False'; ExternalVisible := 'False'; ExternalWritable := 'False'} : Real;
         S_Total { ExternalAccessible := 'False'; ExternalVisible := 'False'; ExternalWritable := 'False'} : Real;
         S_Total_min { ExternalAccessible := 'False'; ExternalVisible := 'False'; ExternalWritable := 'False'} : Real;
         S_Total_max { ExternalAccessible := 'False'; ExternalVisible := 'False'; ExternalWritable := 'False'} : Real;
         P_Total { ExternalAccessible := 'False'; ExternalVisible := 'False'; ExternalWritable := 'False'} : Real;
         P_Total_min { ExternalAccessible := 'False'; ExternalVisible := 'False'; ExternalWritable := 'False'} : Real;
         P_Total_max { ExternalAccessible := 'False'; ExternalVisible := 'False'; ExternalWritable := 'False'} : Real;
         Q_Total { ExternalAccessible := 'False'; ExternalVisible := 'False'; ExternalWritable := 'False'} : Real;
         Q_Total_min { ExternalAccessible := 'False'; ExternalVisible := 'False'; ExternalWritable := 'False'} : Real;
         Q_Total_max { ExternalAccessible := 'False'; ExternalVisible := 'False'; ExternalWritable := 'False'} : Real;
         Cos_L1 { ExternalAccessible := 'False'; ExternalVisible := 'False'; ExternalWritable := 'False'} : Real;
         Cos_L1_min { ExternalAccessible := 'False'; ExternalVisible := 'False'; ExternalWritable := 'False'} : Real;
         Cos_L1_max { ExternalAccessible := 'False'; ExternalVisible := 'False'; ExternalWritable := 'False'} : Real;
         Cos_L2 { ExternalAccessible := 'False'; ExternalVisible := 'False'; ExternalWritable := 'False'} : Real;
         Cos_L2_min { ExternalAccessible := 'False'; ExternalVisible := 'False'; ExternalWritable := 'False'} : Real;
         Cos_L2_max { ExternalAccessible := 'False'; ExternalVisible := 'False'; ExternalWritable := 'False'} : Real;
         Cos_L3 { ExternalAccessible := 'False'; ExternalVisible := 'False'; ExternalWritable := 'False'} : Real;
         Cos_L3_min { ExternalAccessible := 'False'; ExternalVisible := 'False'; ExternalWritable := 'False'} : Real;
         Cos_L3_max { ExternalAccessible := 'False'; ExternalVisible := 'False'; ExternalWritable := 'False'} : Real;
         Cos_Total { ExternalAccessible := 'False'; ExternalVisible := 'False'; ExternalWritable := 'False'} : Real;
         Cos_Total_min { ExternalAccessible := 'False'; ExternalVisible := 'False'; ExternalWritable := 'False'} : Real;
         Cos_Total_max { ExternalAccessible := 'False'; ExternalVisible := 'False'; ExternalWritable := 'False'} : Real;
         S_L1 { ExternalAccessible := 'False'; ExternalVisible := 'False'; ExternalWritable := 'False'} : Real;
         S_L2 { ExternalAccessible := 'False'; ExternalVisible := 'False'; ExternalWritable := 'False'} : Real;
         S_L3 { ExternalAccessible := 'False'; ExternalVisible := 'False'; ExternalWritable := 'False'} : Real;
         S_L1_min { ExternalAccessible := 'False'; ExternalVisible := 'False'; ExternalWritable := 'False'} : Real;
         S_L2_min { ExternalAccessible := 'False'; ExternalVisible := 'False'; ExternalWritable := 'False'} : Real;
         S_L3_min { ExternalAccessible := 'False'; ExternalVisible := 'False'; ExternalWritable := 'False'} : Real;
         S_L1_max { ExternalAccessible := 'False'; ExternalVisible := 'False'; ExternalWritable := 'False'} : Real;
         S_L2_max { ExternalAccessible := 'False'; ExternalVisible := 'False'; ExternalWritable := 'False'} : Real;
         S_L3_max { ExternalAccessible := 'False'; ExternalVisible := 'False'; ExternalWritable := 'False'} : Real;
         P_L1 { ExternalAccessible := 'False'; ExternalVisible := 'False'; ExternalWritable := 'False'} : Real;
         P_L2 { ExternalAccessible := 'False'; ExternalVisible := 'False'; ExternalWritable := 'False'} : Real;
         P_L3 { ExternalAccessible := 'False'; ExternalVisible := 'False'; ExternalWritable := 'False'} : Real;
         P_L1_min { ExternalAccessible := 'False'; ExternalVisible := 'False'; ExternalWritable := 'False'} : Real;
         P_L2_min { ExternalAccessible := 'False'; ExternalVisible := 'False'; ExternalWritable := 'False'} : Real;
         P_L3_min { ExternalAccessible := 'False'; ExternalVisible := 'False'; ExternalWritable := 'False'} : Real;
         P_L1_max { ExternalAccessible := 'False'; ExternalVisible := 'False'; ExternalWritable := 'False'} : Real;
         P_L2_max { ExternalAccessible := 'False'; ExternalVisible := 'False'; ExternalWritable := 'False'} : Real;
         P_L3_max { ExternalAccessible := 'False'; ExternalVisible := 'False'; ExternalWritable := 'False'} : Real;
         Q_L1 { ExternalAccessible := 'False'; ExternalVisible := 'False'; ExternalWritable := 'False'} : Real;
         Q_L2 { ExternalAccessible := 'False'; ExternalVisible := 'False'; ExternalWritable := 'False'} : Real;
         Q_L3 { ExternalAccessible := 'False'; ExternalVisible := 'False'; ExternalWritable := 'False'} : Real;
         Q_L1_min { ExternalAccessible := 'False'; ExternalVisible := 'False'; ExternalWritable := 'False'} : Real;
         Q_L2_min { ExternalAccessible := 'False'; ExternalVisible := 'False'; ExternalWritable := 'False'} : Real;
         Q_L3_min { ExternalAccessible := 'False'; ExternalVisible := 'False'; ExternalWritable := 'False'} : Real;
         Q_L1_max { ExternalAccessible := 'False'; ExternalVisible := 'False'; ExternalWritable := 'False'} : Real;
         Q_L2_max { ExternalAccessible := 'False'; ExternalVisible := 'False'; ExternalWritable := 'False'} : Real;
         Q_L3_max { ExternalAccessible := 'False'; ExternalVisible := 'False'; ExternalWritable := 'False'} : Real;
         E_Active_Rate1_Import { ExternalAccessible := 'False'; ExternalVisible := 'False'; ExternalWritable := 'False'} : Real;
         E_Active_Rate2_Import { ExternalAccessible := 'False'; ExternalVisible := 'False'; ExternalWritable := 'False'} : Real;
         E_Active_Rate1_Export { ExternalAccessible := 'False'; ExternalVisible := 'False'; ExternalWritable := 'False'} : Real;
         E_Active_Rate2_Export { ExternalAccessible := 'False'; ExternalVisible := 'False'; ExternalWritable := 'False'} : Real;
         E_Reactive_Rate1_Import { ExternalAccessible := 'False'; ExternalVisible := 'False'; ExternalWritable := 'False'} : Real;
         E_Reactive_Rate2_Import { ExternalAccessible := 'False'; ExternalVisible := 'False'; ExternalWritable := 'False'} : Real;
         E_Reactive_Rate1_Export { ExternalAccessible := 'False'; ExternalVisible := 'False'; ExternalWritable := 'False'} : Real;
         E_Reactive_Rate2_Export { ExternalAccessible := 'False'; ExternalVisible := 'False'; ExternalWritable := 'False'} : Real;
         E_Apparent_Rate1_Import { ExternalAccessible := 'False'; ExternalVisible := 'False'; ExternalWritable := 'False'} : Real;
         E_Apparent_Rate2_Import { ExternalAccessible := 'False'; ExternalVisible := 'False'; ExternalWritable := 'False'} : Real;
         RTime_Data_Energy { ExternalAccessible := 'False'; ExternalVisible := 'False'; ExternalWritable := 'False'} : Date_And_Time;
         RTime_Data_Value { ExternalAccessible := 'False'; ExternalVisible := 'False'; ExternalWritable := 'False'} : Date_And_Time;
         U_PH_PH_Mod { ExternalAccessible := 'False'; ExternalVisible := 'False'; ExternalWritable := 'False'} : Word;
         U_PH_N_Mod { ExternalAccessible := 'False'; ExternalVisible := 'False'; ExternalWritable := 'False'} : Word;
         I_Mod { ExternalAccessible := 'False'; ExternalVisible := 'False'; ExternalWritable := 'False'} : Word;
         S_Mod { ExternalAccessible := 'False'; ExternalVisible := 'False'; ExternalWritable := 'False'} : Word;
         P_Mod { ExternalAccessible := 'False'; ExternalVisible := 'False'; ExternalWritable := 'False'} : Word;
         Q_Mod { ExternalAccessible := 'False'; ExternalVisible := 'False'; ExternalWritable := 'False'} : Word;
         E_Mod { ExternalAccessible := 'False'; ExternalVisible := 'False'; ExternalWritable := 'False'} : Word;
         f_Mod { ExternalAccessible := 'False'; ExternalVisible := 'False'; ExternalWritable := 'False'} : Word;
         Cos_Mod { ExternalAccessible := 'False'; ExternalVisible := 'False'; ExternalWritable := 'False'} : Word;
         Calculate_Value1 { ExternalAccessible := 'False'; ExternalVisible := 'False'; ExternalWritable := 'False'} : Word;
         Calculate_Value2 { ExternalAccessible := 'False'; ExternalVisible := 'False'; ExternalWritable := 'False'} : Word;
         Calculate_Value3 { ExternalAccessible := 'False'; ExternalVisible := 'False'; ExternalWritable := 'False'} : Word;
         Calculate_Value4 { ExternalAccessible := 'False'; ExternalVisible := 'False'; ExternalWritable := 'False'} : Word;
         Calculate_Value5 { ExternalAccessible := 'False'; ExternalVisible := 'False'; ExternalWritable := 'False'} : Word;
         Calculate_Value6 { ExternalAccessible := 'False'; ExternalVisible := 'False'; ExternalWritable := 'False'} : Word;
         Energy_Meter_Unit { ExternalAccessible := 'False'; ExternalVisible := 'False'; ExternalWritable := 'False'} : Word;
         Rest_Start_Auto { ExternalAccessible := 'False'; ExternalVisible := 'False'; ExternalWritable := 'False'} : Bool;
         Read_Value { ExternalAccessible := 'False'; ExternalVisible := 'False'; ExternalWritable := 'False'} : Bool;
         Connection_Type { ExternalAccessible := 'False'; ExternalVisible := 'False'; ExternalWritable := 'False'} : Int;
         Driver_Error { ExternalAccessible := 'False'; ExternalVisible := 'False'; ExternalWritable := 'False'} : Int;
      END_STRUCT;
      Energy_Counter { ExternalAccessible := 'False'; ExternalVisible := 'False'; ExternalWritable := 'False'} : Struct   // The structure with all energy counter as 64-Bit float values.
         Active_Rate1_Imp_Raw { ExternalAccessible := 'False'; ExternalVisible := 'False'; ExternalWritable := 'False'} : DInt;
         Active_Rate1_Imp_Fine { ExternalAccessible := 'False'; ExternalVisible := 'False'; ExternalWritable := 'False'} : DInt;
         Active_Rate1_Exp_Raw { ExternalAccessible := 'False'; ExternalVisible := 'False'; ExternalWritable := 'False'} : DInt;
         Active_Rate1_Exp_Fine { ExternalAccessible := 'False'; ExternalVisible := 'False'; ExternalWritable := 'False'} : DInt;
         Active_Rate2_Imp_Raw { ExternalAccessible := 'False'; ExternalVisible := 'False'; ExternalWritable := 'False'} : DInt;
         Active_Rate2_Imp_Fine { ExternalAccessible := 'False'; ExternalVisible := 'False'; ExternalWritable := 'False'} : DInt;
         Active_Rate2_Exp_Raw { ExternalAccessible := 'False'; ExternalVisible := 'False'; ExternalWritable := 'False'} : DInt;
         Active_Rate2_Exp_Fine { ExternalAccessible := 'False'; ExternalVisible := 'False'; ExternalWritable := 'False'} : DInt;
         Reactive_Rate1_Imp_Raw { ExternalAccessible := 'False'; ExternalVisible := 'False'; ExternalWritable := 'False'} : DInt;
         Reactive_Rate1_Imp_Fine { ExternalAccessible := 'False'; ExternalVisible := 'False'; ExternalWritable := 'False'} : DInt;
         Reactive_Rate1_Exp_Raw { ExternalAccessible := 'False'; ExternalVisible := 'False'; ExternalWritable := 'False'} : DInt;
         Reactive_Rate1_Exp_Fine { ExternalAccessible := 'False'; ExternalVisible := 'False'; ExternalWritable := 'False'} : DInt;
         Reactive_Rate2_Imp_Raw { ExternalAccessible := 'False'; ExternalVisible := 'False'; ExternalWritable := 'False'} : DInt;
         Reactive_Rate2_Imp_Fine { ExternalAccessible := 'False'; ExternalVisible := 'False'; ExternalWritable := 'False'} : DInt;
         Reactive_Rate2_Exp_Raw { ExternalAccessible := 'False'; ExternalVisible := 'False'; ExternalWritable := 'False'} : DInt;
         Reactive_Rate2_Exp_Fine { ExternalAccessible := 'False'; ExternalVisible := 'False'; ExternalWritable := 'False'} : DInt;
         Apparent_Rate1_Imp_Raw { ExternalAccessible := 'False'; ExternalVisible := 'False'; ExternalWritable := 'False'} : DInt;
         Apparent_Rate1_Imp_Fine { ExternalAccessible := 'False'; ExternalVisible := 'False'; ExternalWritable := 'False'} : DInt;
         Apparent_Rate2_Imp_Raw { ExternalAccessible := 'False'; ExternalVisible := 'False'; ExternalWritable := 'False'} : DInt;
         Apparent_Rate2_Imp_Fine { ExternalAccessible := 'False'; ExternalVisible := 'False'; ExternalWritable := 'False'} : DInt;
      END_STRUCT;
      Time_Between_Update { ExternalAccessible := 'False'; ExternalVisible := 'False'; ExternalWritable := 'False'} : Time := T#0MS;   // The time between the current and the last update of the measurement values.
      Time_Between_Update_Max { ExternalAccessible := 'False'; ExternalVisible := 'False'; ExternalWritable := 'False'} : Time := T#0MS;   // The maximum time between two measurement value updates.
      Time_Stamp_Meas_Values { ExternalAccessible := 'False'; ExternalVisible := 'False'; ExternalWritable := 'False'} : Date_And_Time := DT#1990-01-01-00:00:00;   // The time stamp of the currently available measurement values.
      Error_Location { ExternalAccessible := 'False'; ExternalVisible := 'False'; ExternalWritable := 'False'} : Word := WORD#16#0000;   // The error location or the status of the block. Detailed information in the manual.
      Error_Code { ExternalAccessible := 'False'; ExternalVisible := 'False'; ExternalWritable := 'False'} : DWord := DWORD#16#0000_0000;   // The error code in case of an error of the block, otherwise 0. Detailed information in the manual.
   END_VAR
   VAR_IN_OUT
      HMI_Bits : Struct   // The structure with the feedback of the HMI. Used for the visualization and the connection to the E2M_Visu block.
         Start_Acyclic : Bool;
         Start_Auto : Bool;
         Reset_min_max_Data : Bool;
         Reset_Energy_Meter : Bool;
      END_STRUCT;
      Comm_Resource_Counter { ExternalAccessible := 'False'; ExternalVisible := 'False'; ExternalWritable := 'False'} : Int := 0;   // The counter of the currently used resources from all E2M drivers.
   END_VAR
   VAR
      Read_Data_Record { ExternalAccessible := 'False'; ExternalVisible := 'False'; ExternalWritable := 'False'; S7_SetPoint := 'True'} : RDREC;
      Write_Data_Record { ExternalAccessible := 'False'; ExternalVisible := 'False'; ExternalWritable := 'False'; S7_SetPoint := 'True'} : WRREC;
   END_VAR
   VAR DB_SPECIFIC
      Time_Measurement { ExternalAccessible := 'False'; ExternalVisible := 'False'; ExternalWritable := 'False'; S7_SetPoint := 'True'} : TON_TIME;
      Error_Retry_Timer { ExternalAccessible := 'False'; ExternalVisible := 'False'; ExternalWritable := 'False'; S7_SetPoint := 'True'} : TON_TIME;
      Watchdog { ExternalAccessible := 'False'; ExternalVisible := 'False'; ExternalWritable := 'False'; S7_SetPoint := 'True'} : TON_TIME;
      Reset_Timer { ExternalAccessible := 'False'; ExternalVisible := 'False'; ExternalWritable := 'False'; S7_SetPoint := 'True'} : TON_TIME;
   END_VAR
   VAR
      LREAL_TO_DINT { ExternalAccessible := 'False'; ExternalVisible := 'False'; ExternalWritable := 'False'; S7_SetPoint := 'True'} : "LProcPAC-Conversion";
   END_VAR
   VAR DB_SPECIFIC
      Input_Variables_OK { ExternalAccessible := 'False'; ExternalVisible := 'False'; ExternalWritable := 'False'} : Bool := FALSE;
      HMI_Input_Bits_Connected { ExternalAccessible := 'False'; ExternalVisible := 'False'; ExternalWritable := 'False'} : Bool := FALSE;
      Reset_En_Count_Request { ExternalAccessible := 'False'; ExternalVisible := 'False'; ExternalWritable := 'False'} : Bool := FALSE;
      Reset_Min_Max_Request { ExternalAccessible := 'False'; ExternalVisible := 'False'; ExternalWritable := 'False'} : Bool := FALSE;
      Read_Data_Rec_Request { ExternalAccessible := 'False'; ExternalVisible := 'False'; ExternalWritable := 'False'} : Bool := FALSE;
      Write_Data_Rec_Request { ExternalAccessible := 'False'; ExternalVisible := 'False'; ExternalWritable := 'False'} : Bool := FALSE;
      Start_Acyclic_HMI_Old { ExternalAccessible := 'False'; ExternalVisible := 'False'; ExternalWritable := 'False'} : Bool := FALSE;
      Reset_Energy_HMI_Old { ExternalAccessible := 'False'; ExternalVisible := 'False'; ExternalWritable := 'False'} : Bool := FALSE;
      Reset_Energy_Old { ExternalAccessible := 'False'; ExternalVisible := 'False'; ExternalWritable := 'False'} : Bool := FALSE;
      Reset_Min_Max_HMI_Old { ExternalAccessible := 'False'; ExternalVisible := 'False'; ExternalWritable := 'False'} : Bool := FALSE;
      Reset_Min_Max_Old { ExternalAccessible := 'False'; ExternalVisible := 'False'; ExternalWritable := 'False'} : Bool := FALSE;
      Error_Retry_Timer_Run { ExternalAccessible := 'False'; ExternalVisible := 'False'; ExternalWritable := 'False'} : Bool := FALSE;
      Watchdog_Run { ExternalAccessible := 'False'; ExternalVisible := 'False'; ExternalWritable := 'False'} : Bool := FALSE;
      Reset_Timer_Run { ExternalAccessible := 'False'; ExternalVisible := 'False'; ExternalWritable := 'False'} : Bool := FALSE;
      PE_Request_Reference { ExternalAccessible := 'False'; ExternalVisible := 'False'; ExternalWritable := 'False'} : Byte := BYTE#16#01;
      Sm_State { ExternalAccessible := 'False'; ExternalVisible := 'False'; ExternalWritable := 'False'} : Int := 0;
      Sm_State_Next { ExternalAccessible := 'False'; ExternalVisible := 'False'; ExternalWritable := 'False'} : Int := 0;
      Rd_Rec_Index { ExternalAccessible := 'False'; ExternalVisible := 'False'; ExternalWritable := 'False'} : Int := 0;
      Rd_Rec_Max_Length { ExternalAccessible := 'False'; ExternalVisible := 'False'; ExternalWritable := 'False'} : Int := 0;
      Wr_Rec_Index { ExternalAccessible := 'False'; ExternalVisible := 'False'; ExternalWritable := 'False'} : Int := 0;
      Wr_Rec_Max_Length { ExternalAccessible := 'False'; ExternalVisible := 'False'; ExternalWritable := 'False'} : Int := 0;
      Error_Retry_Counter { ExternalAccessible := 'False'; ExternalVisible := 'False'; ExternalWritable := 'False'} : Int := 0;
      Time_to_update { ExternalAccessible := 'False'; ExternalVisible := 'False'; ExternalWritable := 'False'} : Time := T#0MS;
      HMI_Bits_Internal { ExternalAccessible := 'False'; ExternalVisible := 'False'; ExternalWritable := 'False'} : Struct
         Start_Acyclic { ExternalAccessible := 'False'; ExternalVisible := 'False'; ExternalWritable := 'False'} : Bool := FALSE;
         Start_Auto { ExternalAccessible := 'False'; ExternalVisible := 'False'; ExternalWritable := 'False'} : Bool := FALSE;
         Reset_min_max_Data { ExternalAccessible := 'False'; ExternalVisible := 'False'; ExternalWritable := 'False'} : Bool := FALSE;
         Reset_Energy_Meter { ExternalAccessible := 'False'; ExternalVisible := 'False'; ExternalWritable := 'False'} : Bool := FALSE;
      END_STRUCT;
      Receive_Data_Buffer { ExternalAccessible := 'False'; ExternalVisible := 'False'; ExternalWritable := 'False'} : Array[1..1002] of Byte;
   END_VAR
   VAR
      V_PN_Meas_Data_Res_1 AT Receive_Data_Buffer : Struct   // AT Receive_Data_Buffer : Struct
         Block_Header : Struct
            Block_Type : Word;
            Block_Length : Int;
            Block_Version : Word;
         END_STRUCT;
         Response_Header : Struct
            Service_Request_ID : Byte;
            Request_Reference : Byte;
         END_STRUCT;
         Service_Header_Response : Struct
            Status : Byte;
            Data_Struct_Identifier : Byte;
         END_STRUCT;
         Service_Data_Response : Struct
            Count_Meas_Values : Byte;
            Reserver : Byte;
            Meas_Values_32Bit : Array[1..50] of Struct
               Length_Of_Struct : Int;
               Meas_Data_Struct : Byte;
               Meas_ID_HB : Byte;
               Meas_ID_LB : Byte;
               Meas_Status : Byte;
               Meas_Value : Real;
            END_STRUCT;
         END_STRUCT;
      END_STRUCT;
      V_DP_Meas_Data_Res AT Receive_Data_Buffer : Struct   // AT Receive_Data_Buffer : Struct
         U_L1 : Real;
         U_L2 : Real;
         U_L3 : Real;
         U_L1_L2 : Real;
         U_L2_L3 : Real;
         U_L3_L1 : Real;
         I_L1 : Real;
         I_L2 : Real;
         I_L3 : Real;
         S_L1 : Real;
         S_L2 : Real;
         S_L3 : Real;
         P_L1 : Real;
         P_L2 : Real;
         P_L3 : Real;
         Q_L1 : Real;
         Q_L2 : Real;
         Q_L3 : Real;
         Cos_L1 : Real;
         Cos_L2 : Real;
         Cos_L3 : Real;
         f : Real;
         U_PH_N_Average : Real;
         U_PH_PH_Average : Real;
         I_Average : Real;
         S_Total : Real;
         P_Total : Real;
         Q_Total : Real;
         Cos_Total : Real;
         E_Active_Rate1_Im_HW : DWord;
         E_Active_Rate1_Im_LW : DWord;
         E_Active_Rate2_Im_HW : DWord;
         E_Active_Rate2_Im_LW : DWord;
         E_Active_Rate1_Ex_HW : DWord;
         E_Active_Rate1_Ex_LW : DWord;
         E_Active_Rate2_Ex_HW : DWord;
         E_Active_Rate2_Ex_LW : DWord;
         E_Reactive_Rate1_Im_HW : DWord;
         E_Reactive_Rate1_Im_LW : DWord;
         E_Reactive_Rate2_Im_HW : DWord;
         E_Reactive_Rate2_Im_LW : DWord;
         E_Reactive_Rate1_Ex_HW : DWord;
         E_Reactive_Rate1_Ex_LW : DWord;
         E_Reactive_Rate2_Ex_HW : DWord;
         E_Reactive_Rate2_Ex_LW : DWord;
         E_Apparent_Rate1_Im_HW : DWord;
         E_Apparent_Rate1_Im_LW : DWord;
         E_Apparent_Rate2_Im_HW : DWord;
         E_Apparent_Rate2_Im_LW : DWord;
      END_STRUCT;
      V_DP_Meas_Reset AT Receive_Data_Buffer : Struct   // AT Receive_Data_Buffer : Struct
         Meas_Values : Array[1..47] of DWord;
      END_STRUCT;
      V_DP_Meas_Min_Max AT Receive_Data_Buffer : Struct   // AT Receive_Data_Buffer : Struct
         U_L1_Max : Real;
         U_L2_Max : Real;
         U_L3_Max : Real;
         U_L1_L2_Max : Real;
         U_L2_L3_Max : Real;
         U_L3_L1_Max : Real;
         I_L1_Max : Real;
         I_L2_Max : Real;
         I_L3_Max : Real;
         S_L1_Max : Real;
         S_L2_Max : Real;
         S_L3_Max : Real;
         P_L1_Max : Real;
         P_L2_Max : Real;
         P_L3_Max : Real;
         Q_L1_Max : Real;
         Q_L2_Max : Real;
         Q_L3_Max : Real;
         Cos_L1_Max : Real;
         Cos_L2_Max : Real;
         Cos_L3_Max : Real;
         f_Max : Real;
         U_PH_N_Average_Max : Real;
         U_PH_PH_Average_Max : Real;
         I_Average_Max : Real;
         S_Total_Max : Real;
         P_Total_Max : Real;
         Q_Total_Max : Real;
         Cos_Total_Max : Real;
         U_L1_Min : Real;
         U_L2_Min : Real;
         U_L3_Min : Real;
         U_L1_L2_Min : Real;
         U_L2_L3_Min : Real;
         U_L3_L1_Min : Real;
         I_L1_Min : Real;
         I_L2_Min : Real;
         I_L3_Min : Real;
         S_L1_Min : Real;
         S_L2_Min : Real;
         S_L3_Min : Real;
         P_L1_Min : Real;
         P_L2_Min : Real;
         P_L3_Min : Real;
         Q_L1_Min : Real;
         Q_L2_Min : Real;
         Q_L3_Min : Real;
         Cos_L1_Min : Real;
         Cos_L2_Min : Real;
         Cos_L3_Min : Real;
         f_Min : Real;
         U_PH_N_Average_Min : Real;
         U_PH_PH_Average_Min : Real;
         I_Average_Min : Real;
         S_Total_Min : Real;
         P_Total_Min : Real;
         Q_Total_Min : Real;
         Cos_Total_Min : Real;
      END_STRUCT;
      V_DP_Min_Max_Reset AT Receive_Data_Buffer : Struct   // AT Receive_Data_Buffer : Struct
         Meas_Values : Array[1..58] of DWord;
      END_STRUCT;
      V_PN_Meas_Data_Res_2 AT Receive_Data_Buffer : Struct   // AT Receive_Data_Buffer : Struct
         Block_Header : Struct
            Block_Type : Word;
            Block_Length : Int;
            Block_Version : Word;
         END_STRUCT;
         Response_Header : Struct
            Service_Request_ID : Byte;
            Request_Reference : Byte;
         END_STRUCT;
         Service_Header_Response : Struct
            Status : Byte;
            Data_Struct_Identifier : Byte;
         END_STRUCT;
         Service_Data_Response : Struct
            Count_Meas_Values : Byte;
            Reserver : Byte;
            Meas_Values_32Bit : Array[51..87] of Struct
               Length_Of_Struct : Int;
               Meas_Data_Struct : Byte;
               Meas_ID_HB : Byte;
               Meas_ID_LB : Byte;
               Meas_Status : Byte;
               Meas_Value : Real;
            END_STRUCT;
            Meas_Values_64Bit : Array[88..92] of Struct
               Length_Of_Struct : Int;
               Meas_Data_Struct : Byte;
               Meas_ID_HB : Byte;
               Meas_ID_LB : Byte;
               Meas_Status : Byte;
               Meas_Value_H : DWord;
               Meas_Value_L : DWord;
            END_STRUCT;
         END_STRUCT;
      END_STRUCT;
   END_VAR
   VAR DB_SPECIFIC
      Send_Data_Buffer { ExternalAccessible := 'False'; ExternalVisible := 'False'; ExternalWritable := 'False'} : Array[1..240] of Byte;
   END_VAR
   VAR
      V_PN_Measurement_Data_1 AT Send_Data_Buffer : Struct   // AT Send_Data_Buffer : Struct
         Block_Header : Struct
            Block_Type : Word;
            Block_Length : Int;
            Block_Version : Word;
         END_STRUCT;
         Request_Header : Struct
            Service_Request_ID : Byte;
            Request_Reference : Byte;
         END_STRUCT;
         Service_Header_Request : Struct
            Modifier : Byte;
            Data_Struct_Identifier : Byte;
         END_STRUCT;
         Service_Data_Request : Struct
            Count_Meas_Values : Byte;
            Reserver : Byte;
            Meas_Values : Array[1..50] of Int;
         END_STRUCT;
      END_STRUCT;
      V_DP_Measurement_Data AT Send_Data_Buffer : Struct   // AT Send_Data_Buffer : Struct
         Measurement_Data : Array[1..58] of Struct
            Measurement_ID : Int;
            Measurement_Len : Int;
         END_STRUCT;
      END_STRUCT;
      V_DP_ResetData AT Send_Data_Buffer : Struct   // AT Send_Data_Buffer : Struct
         Command_ID : Array[1..2] of Struct
            Command_ID : Int;
            Command_Len : Int;
            Command_Value : Int;
         END_STRUCT;
      END_STRUCT;
      V_PN_Measurement_Data_2 AT Send_Data_Buffer : Struct   // AT Send_Data_Buffer : Struct
         Block_Header : Struct
            Block_Type : Word;
            Block_Length : Int;
            Block_Version : Word;
         END_STRUCT;
         Request_Header : Struct
            Service_Request_ID : Byte;
            Request_Reference : Byte;
         END_STRUCT;
         Service_Header_Request : Struct
            Modifier : Byte;
            Data_Struct_Identifier : Byte;
         END_STRUCT;
         Service_Data_Request : Struct
            Count_Meas_Values : Byte;
            Reserver : Byte;
            Meas_Values : Array[51..92] of Int;
         END_STRUCT;
      END_STRUCT;
   END_VAR
   VAR_TEMP
      General_Ret_Val : Int;
      Index : Int;
      In_Out_Pointer_Check : Any;
      VIn_Out_Pointer_Check AT In_Out_Pointer_Check : Struct   // AT In_Out_Pointer_Check : Struct
         ID_Type : Word;
         Count : Word;
         DB_Number : Word;
         DB_Offset : DWord;
      END_STRUCT;
   END_VAR
   VAR CONSTANT
      CONNECTION_SINGLE_PHASE : Int := 1;
      CONNECTION_THREE_PHASE : Int := 3;
      PROFINET : Int := 1;
      PROFIBUS : Int := 2;
      RECORD_47_FLEX_ACCESS_MEASUREMENT_INDEX : Int := 47;
      RECORD_PROFIENERGY_INDEX : Word := WORD#16#80A0;
      RECORD_47_WRITE_MEASUREMENT_VALUES_LENGTH : Int := 12;
      RECORD_47_READ_MEASUREMENT_VALUES_LENGTH : Int := 196;
      RECORD_47_WRITE_MINMAX_LEN : Int := 8;
      RECORD_47_READ_MIN_MAX_VALUES_LENGTH : Int := 232;
      RECORD_PE_WRITE_LEN_1 : Int := 112;
      RECORD_PE_WRITE_LEN_2 : Int := 96;
      RECORD_PE_READ_LEN_1 : Int := 512;
      RECORD_PE_READ_LEN_2 : Int := 452;
      RECORD_PE_COUNT_MEAS_1 : Int := 50;
      RECORD_PE_COUNT_MEAS_2 : Int := 42;
      DP_CMD_RESET_MINIMUM_VALUES : Word := WORD#16#EA63;
      DP_CMD_RESET_MAXIMUM_VALUES : Word := WORD#16#EA62;
      DP_CMD_RESET_ENERGY_COUNTER : Word := WORD#16#EA64;
      ERR_LOC_WRITE_MEAS_1 : Word := WORD#16#1311;
      ERR_LOC_WRITE_MEAS_2 : Word := WORD#16#1312;
      ERR_LOC_WRITE_MIN_MAX_VALUES : Word := WORD#16#1313;
      ERR_LOC_WRITE_RES_MIN_MAX : Word := WORD#16#1314;
      ERR_LOC_WRITE_RESET_ENERGY_COUNTER : Word := WORD#16#1315;
      ERR_LOC_READ_MEAS_1 : Word := WORD#16#1321;
      ERR_LOC_READ_MEAS_2 : Word := WORD#16#1322;
      ERR_LOC_READ_MIN_MAX_VALUES : Word := WORD#16#1323;
      ERR_LOC_INVALID_ID : Word := WORD#16#1371;
      ERR_LOC_INVALID_CONNECTION_TYPE : Word := WORD#16#1372;
      ERR_LOC_INVALID_COMM_LIMIT : Word := WORD#16#1373;
      ERR_LOC_INVALID_IO_BYTE : Word := WORD#16#1374;
      ERR_LOC_INVALID_BACKUP_TIME : Word := WORD#16#1375;
      ERR_LOC_INVALID_COMM_COUNTER : Word := WORD#16#1376;
      ERR_LOC_INVALID_COMM_TYPE : Word := WORD#16#1377;
      ERR_LOC_NO_POWER : Word := WORD#16#1381;
      ERR_LOC_PN_INV_BLOCK_1 : Word := WORD#16#1390;
      ERR_LOC_PN_INV_REQ_ID_1 : Word := WORD#16#1391;
      ERR_LOC_PN_INV_REQ_REF_1 : Word := WORD#16#1392;
      ERR_LOC_PN_PE_CMD_FAIL_1 : Word := WORD#16#1393;
      ERR_LOC_PN_INV_DATSTR_1 : Word := WORD#16#1394;
      ERR_LOC_PN_INV_BLOCK_2 : Word := WORD#16#1395;
      ERR_LOC_PN_INVALID_REQUEST_ID_2 : Word := WORD#16#1396;
      ERR_LOC_PN_INV_REQ_REF_2 : Word := WORD#16#1397;
      ERR_LOC_PN_PE_CMD_FAIL_2 : Word := WORD#16#1398;
      ERR_LOC_PN_INV_DATSTR_2 : Word := WORD#16#1399;
      STATUS_IDLE : Word := WORD#16#0000;
      STATUS_WAIT_FOR_RESOURCE : Word := WORD#16#7001;
      STATUS_READ_MEAS : Word := WORD#16#7002;
      STATUS_RESET_MIN_MAX_VALUES : Word := WORD#16#7003;
      STATUS_RESET_ENERGY_COUNTER : Word := WORD#16#7004;
      ERROR_CODE_DEVICE_BUSY : DWord := DWORD#16#DE80_C200;
      ERR_CODE_GENERAL : DWord := DWORD#16#0000_0001;
      ERROR_RETRY_LIMIT : Int := 10;
      DATA_TYPE_WORD : Word := WORD#16#1004;
      DATA_TYPE_INT : Word := WORD#16#1005;
      PN_BLOCK_TYPE_READ : Word := WORD#16#0801;
      PN_REQUEST_ID_GET_MEASUREMENT_VALUES : Byte := BYTE#16#10;
      BIT_RESET_ENERGY_COUNTER : Int := 2;
      BIT_RESET_MINIMUM_VALUES : Int := 0;
      BIT_RESET_MAXIMUM_VALUES : Int := 1;
      TIME_WATCHDOG : Time := T#2S;
      TIME_RETRY_TIMER : Time := T#100MS;
      TIME_RESET_TIMER : Time := T#1S;
      SM_IDLE : Int := 0;
      SM_MEAS_WAIT_RESOURCE : Int := 11;
      SM_WRITE_MEAS_WAIT_RESP : Int := 12;
      SM_READ_MEAS_WAIT_RESP : Int := 13;
      SM_READ_MEAS_WAIT_TIME : Int := 14;
      SM_WRITE_MEAS_PN_WAIT_RESP : Int := 15;
      SM_READ_MEAS_PN_WAIT_RESP : Int := 16;
      SM_READ_MEAS_PN_WAIT_TIME : Int := 17;
      SM_WRITE_MINMAX_WAIT_RESP : Int := 18;
      SM_READ_MINMAX_WAIT_RESP : Int := 19;
      SM_WRITE_MINMAX_DP_RESP : Int := 24;
      SM_READ_MINMAX_DP_WAIT_RESP : Int := 25;
      PE_ID_U_L1 : Int := 1;
      PE_ID_U_L2 : Int := 2;
      PE_ID_U_L3 : Int := 3;
      PE_ID_U_L1_L2 : Int := 4;
      PE_ID_U_L2_L3 : Int := 5;
      PE_ID_U_L3_L1 : Int := 6;
      PE_ID_I_L1 : Int := 7;
      PE_ID_I_L2 : Int := 8;
      PE_ID_I_L3 : Int := 9;
      PE_ID_S_L1 : Int := 10;
      PE_ID_S_L2 : Int := 11;
      PE_ID_S_L3 : Int := 12;
      PE_ID_P_L1 : Int := 13;
      PE_ID_P_L2 : Int := 14;
      PE_ID_P_L3 : Int := 15;
      PE_ID_Q_L1 : Int := 16;
      PE_ID_Q_L2 : Int := 17;
      PE_ID_Q_L3 : Int := 18;
      PE_ID_COS_L1 : Int := 19;
      PE_ID_COS_L2 : Int := 20;
      PE_ID_COS_L3 : Int := 21;
      PE_ID_F : Int := 22;
      PE_ID_U_AVG_L_N : Int := 23;
      PE_ID_U_AVG_L_L : Int := 24;
      PE_ID_I_AVG : Int := 25;
      PE_ID_P_OVERALL : Int := 26;
      PE_ID_Q_OVERALL : Int := 27;
      PE_ID_S_OVERALL : Int := 28;
      PE_ID_COS_OVERALL : Int := 29;
      PE_ID_U_L1_MAX : Int := 30;
      PE_ID_U_L2_MAX : Int := 31;
      PE_ID_U_L3_MAX : Int := 32;
      PE_ID_U_L1_L2_MAX : Int := 33;
      PE_ID_U_L2_L3_MAX : Int := 34;
      PE_ID_U_L3_L1_MAX : Int := 35;
      PE_ID_I_L1_MAX : Int := 36;
      PE_ID_I_L2_MAX : Int := 37;
      PE_ID_I_L3_MAX : Int := 38;
      PE_ID_S_L1_MAX : Int := 39;
      PE_ID_S_L2_MAX : Int := 40;
      PE_ID_S_L3_MAX : Int := 41;
      PE_ID_P_L1_MAX : Int := 42;
      PE_ID_P_L2_MAX : Int := 43;
      PE_ID_P_L3_MAX : Int := 44;
      PE_ID_Q_L1_MAX : Int := 45;
      PE_ID_Q_L2_MAX : Int := 46;
      PE_ID_Q_L3_MAX : Int := 47;
      PE_ID_COS_L1_MAX : Int := 48;
      PE_ID_COS_L2_MAX : Int := 49;
      PE_ID_COS_L3_MAX : Int := 50;
      PE_ID_F_MAX : Int := 51;
      PE_ID_U_AVG_L_N_MAX : Int := 52;
      PE_ID_U_AVG_L_L_MAX : Int := 53;
      PE_ID_I_AVG_MAX : Int := 54;
      PE_ID_P_OVERALL_MAX : Int := 55;
      PE_ID_Q_OVERALL_MAX : Int := 56;
      PE_ID_S_OVERALL_MAX : Int := 57;
      PE_ID_COS_OVERALL_MAX : Int := 58;
      PE_ID_U_L1_MIN : Int := 59;
      PE_ID_U_L2_MIN : Int := 60;
      PE_ID_U_L3_MIN : Int := 61;
      PE_ID_U_L1_L2_MIN : Int := 62;
      PE_ID_U_L2_L3_MIN : Int := 63;
      PE_ID_U_L3_L1_MIN : Int := 64;
      PE_ID_I_L1_MIN : Int := 65;
      PE_ID_I_L2_MIN : Int := 66;
      PE_ID_I_L3_MIN : Int := 67;
      PE_ID_S_L1_MIN : Int := 68;
      PE_ID_S_L2_MIN : Int := 69;
      PE_ID_S_L3_MIN : Int := 70;
      PE_ID_P_L1_MIN : Int := 71;
      PE_ID_P_L2_MIN : Int := 72;
      PE_ID_P_L3_MIN : Int := 73;
      PE_ID_Q_L1_MIN : Int := 74;
      PE_ID_Q_L2_MIN : Int := 75;
      PE_ID_Q_L3_MIN : Int := 76;
      PE_ID_COS_L1_MIN : Int := 77;
      PE_ID_COS_L2_MIN : Int := 78;
      PE_ID_COS_L3_MIN : Int := 79;
      PE_ID_F_MIN : Int := 80;
      PE_ID_U_AVG_L_N_MIN : Int := 81;
      PE_ID_U_AVG_L_L_MIN : Int := 82;
      PE_ID_I_AVG_MIN : Int := 83;
      PE_ID_P_OVERALL_MIN : Int := 84;
      PE_ID_Q_OVERALL_MIN : Int := 85;
      PE_ID_S_OVERALL_MIN : Int := 86;
      PE_ID_COS_OVERALL_MIN : Int := 87;
      PE_ID_E_P_IMP_64 : Int := 88;
      PE_ID_E_P_EXP_64 : Int := 89;
      PE_ID_E_Q_IMP_64 : Int := 90;
      PE_ID_E_Q_EXP_64 : Int := 91;
      PE_ID_E_S_IMP_64 : Int := 92;
   END_VAR
   // Receive_Data_Buffer[1..1000] := BYTE#16#00;
   // Send_Data_Buffer[1..240] := BYTE#16#00;
BEGIN



       // Only check the input variables during the first configuration or
       // until they are correct
       IF (#Input_Variables_OK = FALSE) THEN

           // Also check if a variable is connected to the communication
           // resource counter
           #In_Out_Pointer_Check := #Comm_Resource_Counter;

           // Check each input value for the correct value range
           // The ID of the Energy Meter has to be something bigger than 0
           // as the input bytes can't be negativ
           IF (#ID < 0) THEN

               // Set the error location and the error code for this error
               #Error_Location := #ERR_LOC_INVALID_ID;
               #Error_Code := #ERR_CODE_GENERAL;

               // The First_Byte_I_O_Data of the Energy Meter has to be something bigger than 0
               // as the input bytes can't be negativ
           ELSIF (#First_Byte_I_O_Data < 0) THEN

               // Set the error location and the error code for this error
               #Error_Location := #ERR_LOC_INVALID_IO_BYTE;
               #Error_Code := #ERR_CODE_GENERAL;

               // The available measurement types are only 1 phase measurement with
               // neutral (1), 3 phase measurement without neutral (3) and 3 phase
               // measurement with neutral (4)
           ELSIF ((#Connection_Type <> #CONNECTION_SINGLE_PHASE)
               AND (#Connection_Type <> #CONNECTION_THREE_PHASE)) THEN

               // Set the error location and the error code for this error
               #Error_Location := #ERR_LOC_INVALID_CONNECTION_TYPE;
               #Error_Code := #ERR_CODE_GENERAL;

               // The communication resource limit has to be somehting bigger than 0.
               // Otherwise, there will never be an update of the data
           ELSIF (#Comm_Resource_Limit <= 0) THEN

               // Set the error location and the error code for this error
               #Error_Location := #ERR_LOC_INVALID_COMM_LIMIT;
               #Error_Code := #ERR_CODE_GENERAL;

               // The available communication types are 1 (PROFINET) and 2 (PROFIBUS)
           ELSIF ((#Comm_Type <> #PROFINET)
               AND (#Comm_Type <> #PROFIBUS)) THEN

               // Set the error location and the error code for this error
               #Error_Location := #ERR_LOC_INVALID_COMM_TYPE;
               #Error_Code := #ERR_CODE_GENERAL;

               // A counter for the used resources has to be connected to work
               // If no variable is connected, the DB number and the DB offset
               // are both 0
           ELSIF (((#VIn_Out_Pointer_Check.DB_Number = 0)
               AND (#VIn_Out_Pointer_Check.DB_Offset = 0))
               OR ((#VIn_Out_Pointer_Check.ID_Type <> #DATA_TYPE_WORD)
               AND (#VIn_Out_Pointer_Check.ID_Type <> #DATA_TYPE_INT))
               OR (#VIn_Out_Pointer_Check.Count <> W#16#0001)) THEN

               // Set the error location and the error code for this error
               #Error_Location := #ERR_LOC_INVALID_COMM_COUNTER;
               #Error_Code := #ERR_CODE_GENERAL;

               // No error in the input variables
           ELSE

               // Check if a variable is connected to the HMI Input bits
               // If not, do not try to use these bits and only use internal
               // variables
               #In_Out_Pointer_Check := #HMI_Bits;

               // There is only nothing connected if the DB number is 0 
               // and the DB offset is also 0
               IF ((#VIn_Out_Pointer_Check.DB_Number = 0)
                   AND (#VIn_Out_Pointer_Check.DB_Offset = 0)) THEN

                   // Set the signal, that no structure is connected to the 
                   // HMI input bits
                   #HMI_Input_Bits_Connected := FALSE;
               ELSE
                   // A structure is connected and can be used in the program
                   #HMI_Input_Bits_Connected := TRUE;
               END_IF;

               // Set the signal, that all input variables are OK
               #Input_Variables_OK := TRUE;
           END_IF;

           // The input variables are checked and are OK
       ELSE

           // If a structure is connected to the HMI_Bits input structure
           // copy the values to the internal structure.
           // Otherwise use the initial values of the internal structure.
           IF (#HMI_Input_Bits_Connected = TRUE) THEN

               // Copy the variable to an internal structure
               #HMI_Bits_Internal := #HMI_Bits;
           ELSE
               ; // Use the initial values of the structure variables
           END_IF;

           // Call the instance of the SFB once at the beginning at the code and set its signal during the program
           #Read_Data_Record(REQ := #Read_Data_Rec_Request,
                             ID := #ID, //INT_TO_DWORD(#ID),
                             INDEX := #Rd_Rec_Index,
                             MLEN := #Rd_Rec_Max_Length,
                             RECORD := #Receive_Data_Buffer);

           // Call the instance of the SFB once at the beginning at the code and set its signal during the program
          #Write_Data_Record(REQ := #Write_Data_Rec_Request,
                             ID := #ID,//INT_TO_DWORD(#ID),
                             INDEX := #Wr_Rec_Index,
                             LEN := #Wr_Rec_Max_Length,
                             RECORD := #Send_Data_Buffer);

           // Keep the timer always running to get the time between two updates and during one update
           #Time_Measurement(IN := TRUE,
                             PT := T#21d);

           // Only call the the timer once at the beginning
           #Error_Retry_Timer(IN := #Error_Retry_Timer_Run,
                              PT := #TIME_RETRY_TIMER);

           // Only call the the timer once at the beginning
           #Watchdog(IN := #Watchdog_Run,
                     PT := #TIME_WATCHDOG);

           // Only call the the timer once at the beginning
           #Reset_Timer(IN := #Reset_Timer_Run,
                       PT := #TIME_RESET_TIMER);

           //===========================================================================
           //====== Set the values for the faceplate for E2M ===========================
           //===========================================================================

           // Set the values for the faceplate, to know which values should be displayed
           // First divide by the different measurement types, as different values
           // are activated in the faceplate for different measurement values
           CASE #Connection_Type OF

                   // 1 phase measurement with only L1 and neutral
               #CONNECTION_SINGLE_PHASE:

                   // The values are coded as bit arrays and can be checked in the manual
                   #Driver_Data.U_PH_N_Mod := W#16#1180;
                   #Driver_Data.U_PH_PH_Mod := W#16#0000;
                   #Driver_Data.I_Mod := W#16#1180;
                   #Driver_Data.S_Mod := W#16#1180;
                   #Driver_Data.P_Mod := W#16#1180;
                   #Driver_Data.Q_Mod := W#16#1180;
                   #Driver_Data.E_Mod := W#16#3381;
                   #Driver_Data.f_Mod := W#16#0380;
                   #Driver_Data.Cos_Mod := W#16#1180;

                   // 3 phase measurement with neutral
               #CONNECTION_THREE_PHASE:

                   // The values are coded as bit arrays and can be checked in the manual
                   #Driver_Data.U_PH_N_Mod := W#16#FF80;
                   #Driver_Data.U_PH_PH_Mod := W#16#FF80;
                   #Driver_Data.I_Mod := W#16#FF80;
                   #Driver_Data.S_Mod := W#16#FF80;
                   #Driver_Data.P_Mod := W#16#FF80;
                   #Driver_Data.Q_Mod := W#16#FF80;
                   #Driver_Data.E_Mod := W#16#3381;
                   #Driver_Data.f_Mod := W#16#0380;
                   #Driver_Data.Cos_Mod := W#16#FF80;

               ELSE
                   ; // Not possible, no other measurement type possible
           END_CASE;

           // Check if the minimum and maximum values are calculated or downloaded
           IF ((#Min_Max_Calculated = TRUE)
               AND (#Comm_Type = #PROFIBUS)) THEN

               // Set the signals, which values are calculated
               #Driver_Data.Calculate_Value1 := W#16#FF0F;
               #Driver_Data.Calculate_Value2 := W#16#F66F;
               #Driver_Data.Calculate_Value3 := W#16#B60D;
               #Driver_Data.Calculate_Value4 := W#16#B60D;
               #Driver_Data.Calculate_Value5 := W#16#B60D;
               #Driver_Data.Calculate_Value6 := W#16#BF07;
           ELSE

               // No value is calculated
               #Driver_Data.Calculate_Value1 := W#16#0000;
               #Driver_Data.Calculate_Value2 := W#16#0000;
               #Driver_Data.Calculate_Value3 := W#16#0000;
               #Driver_Data.Calculate_Value4 := W#16#0000;
               #Driver_Data.Calculate_Value5 := W#16#0000;
               #Driver_Data.Calculate_Value6 := W#16#0000;
           END_IF;

           //===========================================================================
           //====== Reset the minimum and maximum values ===============================
           //===========================================================================

           // With a request from the faceplate, reset all minimum and maximum values
           IF (((#HMI_Bits_Internal.Reset_min_max_Data = TRUE)
               AND (#Reset_Min_Max_HMI_Old = FALSE))
               OR ((#Reset_Min_Max = TRUE)
               AND (#Reset_Min_Max_Old = FALSE))) THEN

               // If the values should be calculated, simply reset the values in the code
               IF ((#Min_Max_Calculated = TRUE)
                   AND (#Comm_Type = 2)) THEN

                   // With a positive request, reset all min and max values which are stored
                   // Voltage between phase and neutral
                   #Driver_Data.U_L1_min := #Driver_Data.U_L1;
                   #Driver_Data.U_L1_max := #Driver_Data.U_L1;
                   #Driver_Data.U_L2_min := #Driver_Data.U_L2;
                   #Driver_Data.U_L2_max := #Driver_Data.U_L2;
                   #Driver_Data.U_L3_min := #Driver_Data.U_L3;
                   #Driver_Data.U_L3_max := #Driver_Data.U_L3;

                   // Voltage between phase and phase
                   #Driver_Data.U_L1_L2_min := #Driver_Data.U_L1_L2;
                   #Driver_Data.U_L1_L2_max := #Driver_Data.U_L1_L2;
                   #Driver_Data.U_L2_L3_min := #Driver_Data.U_L2_L3;
                   #Driver_Data.U_L2_L3_max := #Driver_Data.U_L2_L3;
                   #Driver_Data.U_L3_L1_min := #Driver_Data.U_L3_L1;
                   #Driver_Data.U_L3_L1_max := #Driver_Data.U_L3_L1;

                   // Average voltages for both
                   #Driver_Data.U_PH_N_Average_min := #Driver_Data.U_PH_N_Average;
                   #Driver_Data.U_PH_N_Average_max := #Driver_Data.U_PH_N_Average;
                   #Driver_Data.U_PH_PH_Average_min := #Driver_Data.U_PH_PH_Average;
                   #Driver_Data.U_PH_PH_Average_max := #Driver_Data.U_PH_PH_Average;

                   // Current values including average
                   #Driver_Data.I_L1_min := #Driver_Data.I_L1;
                   #Driver_Data.I_L1_max := #Driver_Data.I_L1;
                   #Driver_Data.I_L2_min := #Driver_Data.I_L2;
                   #Driver_Data.I_L2_max := #Driver_Data.I_L2;
                   #Driver_Data.I_L3_min := #Driver_Data.I_L3;
                   #Driver_Data.I_L3_max := #Driver_Data.I_L3;
                   #Driver_Data.I_Average_min := #Driver_Data.I_Average;
                   #Driver_Data.I_Average_max := #Driver_Data.I_Average;

                   // Net frequency
                   #Driver_Data.f_min := #Driver_Data.f;
                   #Driver_Data.f_max := #Driver_Data.f;

                   // Apparent power including overall
                   #Driver_Data.S_L1_min := #Driver_Data.S_L1;
                   #Driver_Data.S_L1_max := #Driver_Data.S_L1;
                   #Driver_Data.S_L2_min := #Driver_Data.S_L2;
                   #Driver_Data.S_L2_max := #Driver_Data.S_L2;
                   #Driver_Data.S_L3_min := #Driver_Data.S_L3;
                   #Driver_Data.S_L3_max := #Driver_Data.S_L3;
                   #Driver_Data.S_Total_min := #Driver_Data.S_Total;
                   #Driver_Data.S_Total_max := #Driver_Data.S_Total;

                   // Reactive power including overall
                   #Driver_Data.Q_L1_min := #Driver_Data.Q_L1;
                   #Driver_Data.Q_L1_max := #Driver_Data.Q_L1;
                   #Driver_Data.Q_L2_min := #Driver_Data.Q_L2;
                   #Driver_Data.Q_L2_max := #Driver_Data.Q_L2;
                   #Driver_Data.Q_L3_min := #Driver_Data.Q_L3;
                   #Driver_Data.Q_L3_max := #Driver_Data.Q_L3;
                   #Driver_Data.Q_Total_min := #Driver_Data.Q_Total;
                   #Driver_Data.Q_Total_max := #Driver_Data.Q_Total;

                   // Effective power including overall
                   #Driver_Data.P_L1_min := #Driver_Data.P_L1;
                   #Driver_Data.P_L1_max := #Driver_Data.P_L1;
                   #Driver_Data.P_L2_min := #Driver_Data.P_L2;
                   #Driver_Data.P_L2_max := #Driver_Data.P_L2;
                   #Driver_Data.P_L3_min := #Driver_Data.P_L3;
                   #Driver_Data.P_L3_max := #Driver_Data.P_L3;
                   #Driver_Data.P_Total_min := #Driver_Data.P_Total;
                   #Driver_Data.P_Total_max := #Driver_Data.P_Total;

                   // Power factor including overall
                   #Driver_Data.Cos_L1_min := #Driver_Data.Cos_L1;
                   #Driver_Data.Cos_L1_max := #Driver_Data.Cos_L1;
                   #Driver_Data.Cos_L2_min := #Driver_Data.Cos_L2;
                   #Driver_Data.Cos_L2_max := #Driver_Data.Cos_L2;
                   #Driver_Data.Cos_L3_min := #Driver_Data.Cos_L3;
                   #Driver_Data.Cos_L3_max := #Driver_Data.Cos_L3;
                   #Driver_Data.Cos_Total_min := #Driver_Data.Cos_Total;
                   #Driver_Data.Cos_Total_max := #Driver_Data.Cos_Total;

                   // Reset also the maximum time between two updates
                   #Time_Between_Update_Max := T#0s;

                   // Set the time, when the min and max values have been reseted
                   #General_Ret_Val := RD_SYS_T(OUT => #Driver_Data.RTime_Data_Value);
               ELSE

                   // Reset also the maximum time between two updates
                   #Time_Between_Update_Max := T#0s;

                   // Set the request to reset the minimum and maximum values
                   #Reset_Min_Max_Request := TRUE;
               END_IF;
           ELSE
               ; // No request for a reset
           END_IF;

           //===========================================================================
           //====== Check for a request to reset the energy counter ====================
           //===========================================================================

           // The energy counter reset can either be triggered from the input of
           // the driver or from the faceplate
           IF (((#Reset_Energy_Counter = TRUE)
               AND (#Reset_Energy_Old = FALSE))
               OR ((#HMI_Bits_Internal.Reset_Energy_Meter = TRUE)
               AND (#Reset_Energy_HMI_Old = FALSE))) THEN

               // Set the request to reset the energy counter
               #Reset_En_Count_Request := TRUE;
           ELSE
               ; // No request detected
           END_IF;

           // Reset the outputs for reseting min and max values in the PAC by using 1
           // As the PAC needs some time, to recognize the positive edge, the outputs can't be 
           // reset directly after setting them
           IF (#Reset_Timer.Q = TRUE) THEN

               // Reset the timer
               #Reset_Timer_Run := FALSE;

               // Reset all control outputs
               //Q[#First_Byte_I_O_Data, #BIT_RESET_MINIMUM_VALUES] := FALSE;
               //Q[#First_Byte_I_O_Data, #BIT_RESET_MAXIMUM_VALUES] := FALSE;
               //Q[#First_Byte_I_O_Data, #BIT_RESET_ENERGY_COUNTER] := FALSE;
               #Driver_Control := #Driver_Control AND 16#0007;
           ELSE
               ; // Timer not finished or not started
           END_IF;

           // Set the state for the state machine
           #Sm_State := #Sm_State_Next;

           //===========================================================================
           //====== Wait for a request to update values or restore energy counter ======
           //===========================================================================

           // Start the state machine for the real functionality of the block
           CASE #Sm_State OF

                   // Wait for the request to update the energy counter or the measurement values
               #SM_IDLE:

                   // Set the state of the block to "Waiting for a new request"
                   #Error_Location := #STATUS_IDLE;

                   // Check for a request to reset the minimum and maximum values
                   IF (#Reset_Min_Max_Request = TRUE) THEN

                       // Reset the request signal
                       #Reset_Min_Max_Request := FALSE;

                       // Read the current time to set the timestamp of the reset of the minimum and maximum values
                       #General_Ret_Val := RD_SYS_T(OUT => #Driver_Data.RTime_Data_Value);

                       // Set the signal to run the reset timer to reset the outputs later
                       #Reset_Timer_Run := TRUE;

                       // The min and max values can only be reset by using 1 with the control bytes
                       // Byte n.0 = reset the minimum values
                       // Byte n.1 = reset the maximum values
                       //Q[#First_Byte_I_O_Data, #BIT_RESET_MINIMUM_VALUES] := TRUE;
                       //Q[#First_Byte_I_O_Data, #BIT_RESET_MAXIMUM_VALUES] := TRUE;
                       #Driver_Control := #Driver_Control OR 16#0003;

                       // Check for a request to reset the energy counter
                   ELSIF (#Reset_En_Count_Request = TRUE) THEN

                       // Reset the request signal
                       #Reset_En_Count_Request := FALSE;

                       // Read the current time to set the timestamp of the reset of the energy counter
                       #General_Ret_Val := RD_SYS_T(OUT => #Driver_Data.RTime_Data_Energy);

                       // Set the signal to run the reset timer to reset the outputs later
                       #Reset_Timer_Run := TRUE;

                       // The energy counter can only be reset by using 1 with the control bytes
                       // Byte n.2 = reset the energy counter
                       //Q[#First_Byte_I_O_Data, #BIT_RESET_ENERGY_COUNTER] := TRUE;
                       #Driver_Control := #Driver_Control OR 16#0001;

                       // Check if the update timer is elapsed ==> then start to update the measurement values
                   ELSIF (((#Automatic_Update = TRUE)
                       OR (#HMI_Bits_Internal.Start_Auto = TRUE)
                       OR ((#HMI_Bits_Internal.Start_Acyclic = TRUE)
                       AND (#Start_Acyclic_HMI_Old = FALSE)))
                       AND (#Comm_Resource_Limit > 0)) THEN

                       // Check the communication type, for the different data record communication
                       // The communication should happen with 1 ==> PROFIenergy
                       IF (#Comm_Type = #PROFINET) THEN

                           // Increase the request reference
                           #PE_Request_Reference := INT_TO_BYTE(BYTE_TO_INT(#PE_Request_Reference) + 1);

                           // The request refence could not be 0
                           IF (#PE_Request_Reference = B#16#00) THEN
                               #PE_Request_Reference := B#16#01;
                           ELSE
                               ; // Request reference valid
                           END_IF;

                           // For the communication with 1, PROFIenergy is used to get the measurement values. Therefore, data record
                           // 0x80A0 is used. Now build this data record, first the Block header.
                           #V_PN_Measurement_Data_1.Block_Header.Block_Type := W#16#0800;
                           #V_PN_Measurement_Data_1.Block_Header.Block_Version := W#16#0100;

                           // Now build the header special for PROFIenergy
                           #V_PN_Measurement_Data_1.Request_Header.Service_Request_ID := #PN_REQUEST_ID_GET_MEASUREMENT_VALUES;
                           #V_PN_Measurement_Data_1.Request_Header.Request_Reference := #PE_Request_Reference;
                           #V_PN_Measurement_Data_1.Service_Header_Request.Modifier := B#16#02;
                           #V_PN_Measurement_Data_1.Service_Header_Request.Data_Struct_Identifier := B#16#01;

                           // Now build the request data
                           #V_PN_Measurement_Data_1.Service_Data_Request.Count_Meas_Values := INT_TO_BYTE(#RECORD_PE_COUNT_MEAS_1);
                           #V_PN_Measurement_Data_1.Service_Data_Request.Meas_Values[PE_ID_U_L1] := 1;
                           #V_PN_Measurement_Data_1.Service_Data_Request.Meas_Values[PE_ID_U_L2] := 2;
                           #V_PN_Measurement_Data_1.Service_Data_Request.Meas_Values[PE_ID_U_L3] := 3;
                           #V_PN_Measurement_Data_1.Service_Data_Request.Meas_Values[PE_ID_U_L1_L2] := 4;
                           #V_PN_Measurement_Data_1.Service_Data_Request.Meas_Values[PE_ID_U_L2_L3] := 5;
                           #V_PN_Measurement_Data_1.Service_Data_Request.Meas_Values[PE_ID_U_L3_L1] := 6;
                           #V_PN_Measurement_Data_1.Service_Data_Request.Meas_Values[PE_ID_I_L1] := 7;
                           #V_PN_Measurement_Data_1.Service_Data_Request.Meas_Values[PE_ID_I_L2] := 8;
                           #V_PN_Measurement_Data_1.Service_Data_Request.Meas_Values[PE_ID_I_L3] := 9;
                           #V_PN_Measurement_Data_1.Service_Data_Request.Meas_Values[PE_ID_S_L1] := 10;
                           #V_PN_Measurement_Data_1.Service_Data_Request.Meas_Values[PE_ID_S_L2] := 11;
                           #V_PN_Measurement_Data_1.Service_Data_Request.Meas_Values[PE_ID_S_L3] := 12;
                           #V_PN_Measurement_Data_1.Service_Data_Request.Meas_Values[PE_ID_P_L1] := 13;
                           #V_PN_Measurement_Data_1.Service_Data_Request.Meas_Values[PE_ID_P_L2] := 14;
                           #V_PN_Measurement_Data_1.Service_Data_Request.Meas_Values[PE_ID_P_L3] := 15;
                           #V_PN_Measurement_Data_1.Service_Data_Request.Meas_Values[PE_ID_Q_L1] := 16;
                           #V_PN_Measurement_Data_1.Service_Data_Request.Meas_Values[PE_ID_Q_L2] := 17;
                           #V_PN_Measurement_Data_1.Service_Data_Request.Meas_Values[PE_ID_Q_L3] := 18;
                           #V_PN_Measurement_Data_1.Service_Data_Request.Meas_Values[PE_ID_COS_L1] := 19;
                           #V_PN_Measurement_Data_1.Service_Data_Request.Meas_Values[PE_ID_COS_L2] := 20;
                           #V_PN_Measurement_Data_1.Service_Data_Request.Meas_Values[PE_ID_COS_L3] := 21;
                           #V_PN_Measurement_Data_1.Service_Data_Request.Meas_Values[PE_ID_F] := 30;
                           #V_PN_Measurement_Data_1.Service_Data_Request.Meas_Values[PE_ID_U_AVG_L_N] := 31;
                           #V_PN_Measurement_Data_1.Service_Data_Request.Meas_Values[PE_ID_U_AVG_L_L] := 32;
                           #V_PN_Measurement_Data_1.Service_Data_Request.Meas_Values[PE_ID_I_AVG] := 33;
                           #V_PN_Measurement_Data_1.Service_Data_Request.Meas_Values[PE_ID_P_OVERALL] := 34;
                           #V_PN_Measurement_Data_1.Service_Data_Request.Meas_Values[PE_ID_Q_OVERALL] := 35;
                           #V_PN_Measurement_Data_1.Service_Data_Request.Meas_Values[PE_ID_S_OVERALL] := 36;
                           #V_PN_Measurement_Data_1.Service_Data_Request.Meas_Values[PE_ID_COS_OVERALL] := 37;

                           // Get the maximum values
                           #V_PN_Measurement_Data_1.Service_Data_Request.Meas_Values[PE_ID_U_L1_MAX] := 40;
                           #V_PN_Measurement_Data_1.Service_Data_Request.Meas_Values[PE_ID_U_L2_MAX] := 41;
                           #V_PN_Measurement_Data_1.Service_Data_Request.Meas_Values[PE_ID_U_L3_MAX] := 42;
                           #V_PN_Measurement_Data_1.Service_Data_Request.Meas_Values[PE_ID_U_L1_L2_MAX] := 43;
                           #V_PN_Measurement_Data_1.Service_Data_Request.Meas_Values[PE_ID_U_L2_L3_MAX] := 44;
                           #V_PN_Measurement_Data_1.Service_Data_Request.Meas_Values[PE_ID_U_L3_L1_MAX] := 45;
                           #V_PN_Measurement_Data_1.Service_Data_Request.Meas_Values[PE_ID_I_L1_MAX] := 46;
                           #V_PN_Measurement_Data_1.Service_Data_Request.Meas_Values[PE_ID_I_L2_MAX] := 47;
                           #V_PN_Measurement_Data_1.Service_Data_Request.Meas_Values[PE_ID_I_L3_MAX] := 48;
                           #V_PN_Measurement_Data_1.Service_Data_Request.Meas_Values[PE_ID_S_L1_MAX] := 49;
                           #V_PN_Measurement_Data_1.Service_Data_Request.Meas_Values[PE_ID_S_L2_MAX] := 50;
                           #V_PN_Measurement_Data_1.Service_Data_Request.Meas_Values[PE_ID_S_L3_MAX] := 51;
                           #V_PN_Measurement_Data_1.Service_Data_Request.Meas_Values[PE_ID_P_L1_MAX] := 52;
                           #V_PN_Measurement_Data_1.Service_Data_Request.Meas_Values[PE_ID_P_L2_MAX] := 53;
                           #V_PN_Measurement_Data_1.Service_Data_Request.Meas_Values[PE_ID_P_L3_MAX] := 54;
                           #V_PN_Measurement_Data_1.Service_Data_Request.Meas_Values[PE_ID_Q_L1_MAX] := 55;
                           #V_PN_Measurement_Data_1.Service_Data_Request.Meas_Values[PE_ID_Q_L2_MAX] := 56;
                           #V_PN_Measurement_Data_1.Service_Data_Request.Meas_Values[PE_ID_Q_L3_MAX] := 57;
                           #V_PN_Measurement_Data_1.Service_Data_Request.Meas_Values[PE_ID_COS_L1_MAX] := 58;
                           #V_PN_Measurement_Data_1.Service_Data_Request.Meas_Values[PE_ID_COS_L2_MAX] := 59;
                           #V_PN_Measurement_Data_1.Service_Data_Request.Meas_Values[PE_ID_COS_L3_MAX] := 60;

                           // Configure the data record number and the length of the data record
                           #Wr_Rec_Index := WORD_TO_INT(#RECORD_PROFIENERGY_INDEX);
                           #Wr_Rec_Max_Length := #RECORD_PE_WRITE_LEN_1;
                           #V_PN_Measurement_Data_1.Block_Header.Block_Length := #Wr_Rec_Max_Length - 4;

                           // The PAC is connected with 2
                       ELSIF (#Comm_Type = 2) THEN

                           // Configure the data record to write the values to the SENTRON PAC, which should be provided in this data record
                           // As there are too many values which should be provided and the maximum length of the data record is 240 byte,
                           // the reading of the measurement values is divided into two cycles, if the min and max values should not be
                           // calculated in the FB

                           // In the first reading, get the current values from the SENTRON PAC.
                           // ==> Configure the data record, to get the values by using the block reading of more values with one command

